(*
version 1.0	6 oct 2006
programmer 	hugo
tested by		tobias

findB_noNum searches str backwards and returns the last position which is not a number.
a number is characterized by a letter "0..9" or "."

*)
pt := ADR(str) + LEN(str) - 1;
findB_nonum := 0;
FOR pos := LEN(str) TO 1 BY -1 DO;
	IF NOT((PT^ > 47 AND PT^ < 58) OR PT^ = 46) THEN
		findB_nonum := pos;
		RETURN;
	END_IF;
	PT := PT - 1;
END_FOR;
END_FUNCTION

(* POU findB_Num, ST *)
FUNCTION findB_Num : INT
VAR_INPUT
	str : STRING;
END_VAR
VAR
	pos: INT;
	pt : POINTER TO BYTE;
END_VAR

(*
version 1.0	6 oct 2006
programmer 	hugo
tested by		tobias

findB_Num searches str backward and returns the last position of a number
a number is characterized by a letter "0..9" or "."

*)
pt := ADR(str) + LEN(str) - 1;
findB_Num := 0;
FOR pos := LEN(str) TO 1 BY -1 DO;
	IF (PT^ > 47 AND PT^ < 58) OR PT^ = 46 THEN
		findB_Num := pos;
		RETURN;
	END_IF;
	PT := PT - 1;
END_FOR;
END_FUNCTION

(* POU F_Lamp, ST *)
FUNCTION_BLOCK F_Lamp
VAR_INPUT
	SWITCH : BOOL;
	DIMM : BYTE := 255;
	Rst : BOOL;
END_VAR
VAR_OUTPUT
	Lamp : BYTE;
	ontime : REAL;
	cycles : REAL;
	Status : BYTE;
END_VAR
VAR_INPUT CONSTANT
	T_no_Dimm : REAL := 100;
	T_Maintenance : REAL := 15000;
END_VAR
VAR
	runtime : ontime;
	maintenance: BOOL;
END_VAR

(*
version 1.1	8 Feb 2007
programmer 	hugo
tested by		tobias

F_Lamp is an interface to flourescent lamps. its main purpose is to protect flourescent lamps from dimming within the first T_NO_DIMM Time.
If Flourescent Lamps are dimmed during the first 100 hours the lifetime of the lamp is reduced dramatically.
The interface also counts ontime and cycles of the lamp for maintanance purposes.

*)
IF rst THEN
	runtime.rst := TRUE;
	runtime();
	runtime.rst := FALSE;
	ontime := runtime.ontime;
	cycles := runtime.cycles;
	maintenance := FALSE;
ELSE
	runtime(in := Switch);
	ontime := runtime.ontime;
	cycles := runtime.cycles;
END_IF;

IF NOT maintenance AND runtime.ontime >= T_maintenance AND T_Maintenance > 0 THEN
	status := 120;
	maintenance := TRUE;
ELSIF Switch THEN
	IF runtime.ontime < T_no_Dimm THEN
		Lamp := 255;
		STATUS := 111;
	ELSE
		Lamp := DIMM;
		status := 112;
	END_IF;
ELSE
	lamp := 0;
	status := 110;
END_IF;
END_FUNCTION_BLOCK

(* POU F_lin, ST *)
FUNCTION F_lin : REAL
VAR_INPUT
	X : REAL;
	A : REAL;
	B : REAL;
END_VAR
VAR
END_VAR

(*
version 1.0	1 sep 2006
programmer 	hugo
tested by		tobias

this function calculates the linear equation f_lin = a*x + b

*)
F_lin := A * X + B;
END_FUNCTION

(* POU F_Lin2, ST *)
FUNCTION F_Lin2 : REAL
VAR_INPUT
	X : REAL;
	X1: REAL;
	Y1 : REAL;
	X2 : REAL;
	Y2 : REAL;
END_VAR
VAR

END_VAR

(*
version 1.0	1 jan 2007
programmer 	hugo
tested by		tobias

this function calculates the linear equation f_lin = a*x + b given by two points x1/y1 and x2/y2.

*)
F_Lin2 := (Y2 - Y1) / (X2 - X1) * X + (Y1 * X1 - Y2 * X1) / (X2 - X1) + Y1;
END_FUNCTION

(* POU F_power, ST *)
FUNCTION F_power : REAL
VAR_INPUT
	a : REAL;
	x : REAL;
	n : REAL;
END_VAR
VAR
END_VAR

(*
version 1.0	1 sep 2006
programmer 	hugo
tested by		tobias

this function calculates the power equation f_power = a*x^n

*)
f_power := a * EXPT(X,N);
END_FUNCTION

(* POU F_quad, ST *)
FUNCTION F_quad : REAL
VAR_INPUT
	X : REAL;
	A : REAL;
	B : REAL;
	C : REAL;
END_VAR
VAR
END_VAR

(*
version 1.0	1 sep 2006
programmer 	hugo
tested by		tobias

this function calculates the quadratic equation f_lin = a*x + b

*)
F_quad := a * X * X + B * X + C;
END_FUNCTION

(* POU F_to_C, ST *)
FUNCTION F_to_C : REAL
VAR_INPUT
	fahrenheit : REAL;
END_VAR
VAR
END_VAR

(*
version 1.0	4 aug 2006
programmer 	hugo
tested BY		tobias

this FUNCTION converts fahrenheit TO celsius

executioin TIME on wago 750-841 = 15us
*)
F_to_C := (fahrenheit -32) / 1.8;
END_FUNCTION

(* POU F_to_OM, ST *)
FUNCTION F_to_OM : REAL
VAR_INPUT
	F : REAL;
END_VAR
VAR
END_VAR

(*
version 1.0	22 jan 2007
programmer 	hugo
tested by		tobias

this function converts frequency to Omega F
Omega = 2*PI*F
*)
F_to_OM := PI2 * F;
END_FUNCTION

(* POU F_to_PT, ST *)
FUNCTION F_to_PT : TIME
VAR_INPUT
	F : REAL;
END_VAR
VAR
END_VAR

(*
version 1.0	4 aug 2006
programmer 	hugo
tested by		tobias

this function converts frequency to periode time  
*)
F_to_PT := DWORD_TO_TIME(REAL_TO_DWORD(1/F*1000));
END_FUNCTION

(* POU fact, ST *)
FUNCTION fact : INT
VAR_INPUT
	X : INT;
END_VAR
VAR
	i: INT;
END_VAR

(*
version 1.1	4 mar 2007
programmer 	hugo
tested by		tobias

this function calculates the factorial of x
this simple factorial only calculates factorials for inputs up to 7
if the input is negative or higher then 7 the output will be -1.

*)
IF x >= 0 AND x < 8 THEN
	fact := 1;
	i := 1;
	WHILE i <= x DO
		fact := fact * i;
		i := i + 1;
	END_WHILE;
ELSE
	fact := -1;
END_IF;

(* revision history
hm 4.3.2007	rev 1.1
	changed a critical error where while loop was indefinite.

*)
END_FUNCTION

(* POU FF_D2E, ST *)
FUNCTION_BLOCK FF_D2E
VAR_INPUT
	D0 : BOOL := 0;
	D1 : BOOL := 0;
	CLK : BOOL;
	RST : BOOL := 0;
END_VAR
VAR_OUTPUT
	Q0 : BOOL := 0;
	Q1 : BOOL := 0;
END_VAR
VAR
	edge : BOOL;
END_VAR

(*
version 1.0	4 aug 2006
programmer 	hugo
tested by		tobias

dual D-type flip flop with reset and rising clock trigger

executioin TIME on wago 750-841 = 6us
*)
IF rst THEN
	Q0 := FALSE;
	Q1 := FALSE;
ELSE
	IF clk AND NOT edge THEN
		Q0 := D0;
		Q1 := D1;
	END_IF;
END_IF;
edge := CLK;
END_FUNCTION_BLOCK

(* POU FF_D4E, ST *)
FUNCTION_BLOCK FF_D4E
VAR_INPUT
	D0 : BOOL := 0;
	D1 : BOOL := 0;
	D2 : BOOL := 0;
	D3 : BOOL := 0;
	CLK : BOOL;
	RST : BOOL := 0;
END_VAR
VAR_OUTPUT
	Q0 : BOOL := 0;
	Q1 : BOOL := 0;
	Q2 : BOOL := 0;
	Q3 : BOOL := 0;
END_VAR
VAR
	edge : BOOL;
END_VAR


(*
version 1.0	4 aug 2006
programmer 	hugo
tested by		tobias

quad D-type flip flop with reset and rising clock trigger

executioin TIME on wago 750-841 = 6us
*)
IF rst THEN
	Q0 := FALSE;
	Q1 := FALSE;
	Q2 := FALSE;
	Q3 := FALSE;
ELSE
	IF clk AND NOT edge THEN
		Q0 := D0;
		Q1 := D1;
		Q2 := D2;
		Q3 := D3;
	END_IF;
END_IF;
edge := CLK;
END_FUNCTION_BLOCK

(* POU FF_DRE, ST *)
FUNCTION_BLOCK FF_DRE
VAR_INPUT
	SET : BOOL;
	D : BOOL;
	CLK : BOOL;
	RST : BOOL;
END_VAR
VAR_OUTPUT
	Q : BOOL := 0;
END_VAR
VAR
	edge : BOOL;
END_VAR


(*
version 1.0	4 aug 2006
programmer 	hugo
tested by		tobias

D-type flip flop with set, reset and rising clock trigger
executioin TIME on wago 750-841 = 8us
*)
IF rst THEN
	Q := FALSE;
ELSIF set AND NOT rst THEN
	Q := TRUE;
ELSE
	IF clk AND NOT edge THEN Q := D; END_IF;
END_IF;
edge := CLK;
END_FUNCTION_BLOCK

(* POU FF_JKE, ST *)
FUNCTION_BLOCK FF_JKE
VAR_INPUT
	SET : BOOL;
	J : BOOL;
	CLK : BOOL;
	K : BOOL;
	RST : BOOL;
END_VAR
VAR_OUTPUT
	Q : BOOL := 0;
END_VAR
VAR
	edge : BOOL;
END_VAR


(*
version 1.0	4 aug 2006
programmer 	hugo
tested by		tobias

JK-type flip flop with set, reset and rising clock trigger
set and reset are asynchron while the FF is rising edge triggered
J=0 and K=0 and CLK >>> no action
J=1 and K=0 and CLK >>> output = 1
J=0 and K=1 and CLK >>> output = 0
J=1 and K=1 and CLK >>> toggle output

executioin TIME on wago 750-841 = 8us
*)
IF rst THEN
	Q := FALSE;
ELSIF set AND NOT rst THEN
	Q := TRUE;
ELSE
	IF clk AND NOT edge THEN
		IF J AND NOT K THEN Q := TRUE;
		ELSIF K AND NOT J THEN Q := FALSE;
		ELSIF K AND J THEN Q:= NOT Q;
		END_IF;
	END_IF;
END_IF;
edge := CLK;
END_FUNCTION_BLOCK

(* POU FIFO_16, ST *)
FUNCTION_BLOCK FIFO_16
VAR_INPUT
	Din : DWORD;
	WR : BOOL;
	E : BOOL;
	RST : BOOL;
END_VAR
VAR_OUTPUT
	Dout : DWORD := 0;
	empty : BOOL := TRUE;
	full : BOOL := FALSE;
END_VAR
VAR
	fifo : ARRAY[0..15] OF DWORD;
	NW : INT := 0;
	NR : INT := 0;
	top : INT := 15;
END_VAR

(*
	version 1.0	4 aug 2006
	programmer 	hugo
	tested by		tobias

16 Dword FIFO memory
*)
IF rst THEN
	(* asynchronous reset for the fifo *)
	NW := 0;
	NR := 0;
	Dout := 0;
	empty := TRUE;
	full := FALSE;
ELSIF WR AND E AND NOT full THEN
	(* write action *)
	fifo[NW] := Din;
	IF NW = top THEN NW := 0; ELSE NW := NW + 1; END_IF
	IF NW = NR THEN full := TRUE; END_IF
	empty := FALSE;
ELSIF NOT WR AND E AND NOT empty THEN
	(* read from stack *)
	Dout := fifo[NR];
	IF NR = top THEN NR := 0; ELSE NR := NR + 1; END_IF;
	IF NR = NW THEN empty := TRUE; END_IF;
	full := FALSE;
END_IF;
END_FUNCTION_BLOCK

(* POU FIFO_32, ST *)
FUNCTION_BLOCK FIFO_32
VAR_INPUT
	Din : DWORD;
	WR : BOOL;
	E : BOOL;
	RST : BOOL;
END_VAR
VAR_OUTPUT
	Dout : DWORD := 0;
	empty : BOOL := TRUE;
	full : BOOL := FALSE;
END_VAR
VAR
	fifo : ARRAY[0..31] OF DWORD;
	NW : INT := 0;
	NR : INT := 0;
	top : INT := 31;
END_VAR

(*
	version 1.0	4 aug 2006
	programmer 	hugo
	tested by		tobias

32 Dword FIFO memory
*)
IF rst THEN
	(* asynchronous reset for the fifo *)
	NW := 0;
	NR := 0;
	Dout := 0;
	empty := TRUE;
	full := FALSE;
ELSIF WR AND E AND NOT full THEN
	(* write action *)
	fifo[NW] := Din;
	IF NW = top THEN NW := 0; ELSE NW := NW + 1; END_IF
	IF NW = NR THEN full := TRUE; END_IF
	empty := FALSE;
ELSIF NOT WR AND E AND NOT empty THEN
	(* read from stack *)
	Dout := fifo[NR];
	IF NR = top THEN NR := 0; ELSE NR := NR + 1; END_IF;
	IF NR = NW THEN empty := TRUE; END_IF;
	full := FALSE;
END_IF;
END_FUNCTION_BLOCK

(* POU find_nonum, ST *)
FUNCTION find_nonum : INT
VAR_INPUT
	str : STRING;
END_VAR
VAR
	pos: INT;
	pt : POINTER TO BYTE;
END_VAR

(*
version 1.0	6 oct 2006
programmer 	hugo
tested by		tobias

find_noNum searches str and returns the first position which is not a number.
a number is characterized by a letter "0..9" or "."

*)
pt := ADR(str);
find_nonum := 0;
FOR pos := 1 TO LEN(str) DO;
	IF NOT((PT^ > 47 AND PT^ < 58) OR PT^ = 46) THEN
		find_nonum := pos;
		RETURN;
	END_IF;
	PT := PT + 1;
END_FOR;
END_FUNCTION

(* POU find_Num, ST *)
FUNCTION find_Num : INT
VAR_INPUT
	str : STRING;
END_VAR
VAR
	pos: INT;
	pt : POINTER TO BYTE;
END_VAR

(*
version 1.0	6 oct 2006
programmer 	hugo
tested by		tobias

find_Num searches str and returns the starting position of a number
a number is characterized by a letter "0..9" or "."

*)
pt := ADR(str);
find_Num := 0;
FOR pos := 1 TO LEN(str) DO;
	IF (PT^ > 47 AND PT^ < 58) OR PT^ = 46 THEN
		find_Num := pos;
		RETURN;
	END_IF;
	PT := PT + 1;
END_FOR;
END_FUNCTION

(* POU FindB, ST *)
FUNCTION FindB : INT
VAR_INPUT
	str1 : STRING;
	str2 : STRING;
END_VAR
VAR
	pos: INT;
	size: INT;
	length: INT;
END_VAR

(*
version 1.0	6 oct 2006
programmer 	hugo
tested by		tobias

the function find searches an str1 for the presence of str2 and returns the first position of str1 of the last presence in instring.
the function is similar to find except it searches from the right to left.
 a 0 is returned if the string is not found.

*)
size := LEN(str1);
length := LEN(str2);
FOR pos := size TO 1 BY -1 DO
	IF MID(str1,length,pos) = str2 THEN
		FindB := pos;
		RETURN;
	END_IF;
END_FOR;
END_FUNCTION

(* POU floor, ST *)
FUNCTION floor : INT
VAR_INPUT
	X : REAL;
END_VAR
VAR
END_VAR


(*
version 1.0	7 feb 2007
programmer 	hugo
tested by		tobias

This is a rounding function which returns the biggest possible integer which is less or equal to X.
floor(3.14) = 3
floor(-3.14) = 4

*)
floor := TRUNC(X);
IF floor > X THEN
	floor := floor - 1;
END_IF;
END_FUNCTION

(* POU fract, ST *)
FUNCTION fract : REAL
VAR_INPUT
	input : REAL;
END_VAR
VAR
END_VAR
VAR
END_VAR

(*
version 1.0	4 aug 2006
programmer 	hugo
tested by		tobias

this function returns the fraction of a real number
fract(3.14) = 0.14

execution time on wago 750 - 841 =  17  us
*)
fract := input - TRUNC(input);
END_FUNCTION

(* POU FT_avg, ST *)
FUNCTION_BLOCK FT_avg
VAR_INPUT
	in : REAL;
	en : BOOL;
	N : INT;
	rst : BOOL;
END_VAR
VAR_OUTPUT
	avg : REAL;
END_VAR
VAR
	buff : delay;
	i: INT;
	init : BOOL;
END_VAR

(*
version 1.1	7 jan 2007
programmer 	hugo
tested by		tobias

this function calculates the average over n samples from a sequential input
the input values are shifted into an N deep buffer and the avg of this buffer is diplayed at anytime on the output.
a rst will load the buffer with the current in value..

*)
(* limit n to a max of 32 because delay can do max 32 cycles *)
IF N > 32 THEN
	buff.n := 32;
ELSIF N < 0 THEN
	Buff.n := 0;
ELSE
	buff.n := N;
END_IF;

IF NOT init THEN
	FOR i := 1 TO N DO
		buff(in := in);
	END_FOR;
	avg := in;
	init := TRUE;
ELSIF rst THEN
	FOR i := 1 TO N DO
		buff(in := in);
	END_FOR;
	avg := in;
ELSIF en THEN
	buff(in := in);
	avg := avg + (in - buff.out)/N;
END_IF;

(* revision history

hm	7.1.2007	rev 1.1
	chaged rst logic to load the buffer with the actual input value instead of 0.
	added en input to allow better control of signal flow
	added init to load the buffer with inat startup to avoid rampup at beginning.
	deleted unused variable cnt.
*)
END_FUNCTION_BLOCK

(* POU FT_deriv, ST *)
FUNCTION_BLOCK FT_deriv
VAR_INPUT
	in : REAL;
	K : REAL := 1;
	run : BOOL := 1;
END_VAR
VAR_OUTPUT
	out : REAL;
END_VAR
VAR
	old: REAL;
	tx: TIME;
	last: TIME;
	init: BOOL;
END_VAR


(*
version 1.1	3 jan 2007
programmer 	hugo
tested by		tobias

FT_deriv calculates the derivate over the signal "in" with Faktor "K".
a run input enables or stops the calculation, if left unconnected its true and therfore the calculation is executed.
if K is not specified the default is 1.

*)
tx := TIME();
IF NOT init THEN
	init := TRUE;
	old := in;
	last := tx;
END_IF;
IF run THEN
	out := (in - old) / TIME_TO_REAL(tx - last) * 1000 * K;
ELSE
	out := 0;
END_IF;
old := in;
last := tx;

(*
hm 3.1.2007	rev 1.1
	added init code for startup
	set the default for K to 1

*)
END_FUNCTION_BLOCK

(* POU FT_IMP, ST *)
FUNCTION_BLOCK FT_IMP
VAR_INPUT
	in : REAL;
	T : TIME;
	K : REAL := 1;
END_VAR
VAR_OUTPUT
	out : REAL;
END_VAR
VAR
	t1 : FT_PT1;
END_VAR

(*
version 1.1	3 Jan 2007
programmer 	hugo
tested by		tobias

FT_IMP is 	an impulse filter (high pass filter) with the time T and factor K.
 
*)
T1(in:= in, T:=T);
out := (in - t1.out) * K;

(*
hm 3.1.2007	rev 1.1
	added factor K

*)
END_FUNCTION_BLOCK

(* POU FT_PT1, ST *)
FUNCTION_BLOCK FT_PT1
VAR_INPUT
	in : REAL;
	T : TIME;
	K : REAL := 1;
END_VAR
VAR_OUTPUT
	out : REAL;
END_VAR
VAR
	last : TIME;
	tx: TIME;
	init: BOOL;
END_VAR

(*
version 1.3	27 feb 2007
programmer 	hugo
tested by		tobias

FT_PT1 is an low pass filter with a programmable time T and faktor K.
 
*)
tx := TIME();
IF NOT init THEN
	last := tx;
	init := TRUE;
ELSIF T = t#0s THEN
	out := in;
ELSE
	out := out + (in * K - out) * TIME_TO_REAL(Tx - last) / TIME_TO_REAL(T);
END_IF;
last := tx;

(*
hm 1.1.2007	rev 1.1
	corrected error while startup value was not correct
	for very small time values real output would run out of range.

hm 3.1.2007	rev 1.2
	corrected an error for falling edge failures.
	added output faktor K.

hm 27. 2. 2007	rev 1.3
	output will be input during init for definitive startup condition.
*)
END_FUNCTION_BLOCK

(* POU FT_INT, ST *)
FUNCTION_BLOCK FT_INT
VAR_INPUT
	in : REAL;
	K : REAL := 1;
	run : BOOL := 1;
	rst: BOOL := 0;
	out_min : REAL := -1000;
	out_max : REAL := 1000;
END_VAR
VAR_OUTPUT
	Out : REAL;
	ET: TIME;
END_VAR
VAR
	last: TIME;
	in_last : REAL;
	tx: TIME;
	init: BOOL;
END_VAR


(*
version 1.2	15 jan 2007
programmer 	hugo
tested by		tobias

FT_int is an integrator with input IN and factor K.
integration is only done while run = true, if run is false integration is stopped and the out remains at the last value.
if run is left unconnected, run is considered true by the function block.
the output ET will display the total integration time from last reset.
a rst input will reset output and the timer ET to 0.
the out_min and out_max values can be set to ,imit the output value range. 
out _min is preset to -1000 and out_max is preset to 1000.
the default for K is 1.

 
*)
last := tx;
tx := TIME();
IF rst OR NOT init THEN
	out := 0;
	ET := t#0s;
	init := TRUE;
	last := tx;
ELSIF run THEN
	out := out + (in + in_last)/2 * TIME_TO_DINT(Tx-last) * K / 1000;
	IF out < out_min THEN out := out_min; ELSIF out > out_max THEN out := out_max; END_IF;
	et := et + Tx - last;
END_IF;
in_last := in;

(*
hm 13.12.2006	rev 1.1
changed to "trapezregel" which increases accuracy
before out := out + in * time new: out := out + (in + in_last) / 2 * time

hm 15.1.2007		rev 1.2
added default for k to be 1.
*)
END_FUNCTION_BLOCK

(* POU FT_min_max, ST *)
FUNCTION_BLOCK FT_min_max
VAR_INPUT
	in : REAL;
	rst : BOOL;
END_VAR
VAR_OUTPUT
	mx : REAL;
	mn : REAL;
END_VAR
VAR
	init: BOOL;
END_VAR

(*
version 1.0	1 sep 2006
programmer 	hugo
tested by		tobias

this function block stores the min and max value of an input signal.
when rst is true the mn and mx outputs are set to the in value.
when a rst is never active the function autoresets to the in value at startup.
since the input might not be present at first cycle the mn and mx are set during second cycle.

*)
IF rst OR NOT init THEN
	mn := in;
	mx := in;
	init := 1;
ELSIF in < mn THEN mn := in;
ELSIF in > mx THEN mx := in;
END_IF;
END_FUNCTION_BLOCK

(* POU FT_PID, ST *)
FUNCTION_BLOCK FT_PID
VAR_INPUT
	actual, set_point, offset, manual_in : REAL;
	Manual : BOOL;
	rst : BOOL := FALSE;
	int_band : REAL := 100;
END_VAR
VAR_INPUT
	KP : REAL := 1.0;
	TN : REAL := 1.0;
	TV : REAL := 1.0;
	limit_L : REAL := -1000;
	limit_H : REAL := 1000;
END_VAR
VAR_OUTPUT
	Y : REAL;
	LIM, overflow : BOOL;
END_VAR
VAR
	integ : FT_INT;
	deriv : FT_deriv;
	diff: REAL;
END_VAR

(*
version 1.3	3 mar 2007
programmer 	hugo
tested by		tobias

FT_PID is a pid controller with manual functionality.
The PID controller works according to the fomula Y = KP * ( e + 1/TN * INTEG(e) + TV *DERIV(e)) + offset, while e = set_point - actual.
a rst will reset all internal data, while a switch to manual will cause the controller to follow the function Y = manual_in + offset.
limit_h and Limit_l set the possible output range of Y.
the output flags lim will signal that the output limits are active and overflow will signal that the integrator has reached the max or min limit.  

since rev 1.1 the "trapezregel is used for more accuracy.
rev 1.2 added selective integratin which means the integrative component is only active within a small range of the target value 
this avoids the integrator to go to limits while an input setpoint change happened and is only causing overshoots.
the int_band is by default 100 which means the int is active all the time and if set to for example to 0.1 the integrator is only active
while the input is between 0.9 and 1.1 of the set_point value.

default values for KP = 1, TN = 1, TV = 1, LIMIT_L = -1000, LIMIT_H = +1000.
*)
IF rst OR KP = 0 THEN
	y := offset;
	integ(rst := 1);
	integ.rst := 0;
ELSIF manual THEN
	Y := manual_in + offset;
	integ(rst := 1);
	integ.rst := 0;
ELSE
	(* calcualtion of the actual PID values *)
	diff := set_point - actual;

	(* integrator is only called if TN > 0 and input is within int_band othewrwise it is disabled *)
	IF TN > 0 AND actual > set_point - int_band AND actual < set_point + int_band THEN
		integ(in := diff, K := 1/TN, out_min := (limit_L - offset) / KP, out_max := (limit_H - offset) / KP);
	ELSE
		integ(rst := 1);
		integ.rst := 0;
	END_IF;
	deriv(in := diff, K := TV);

	(* check if integrator has reached the allowed limits and set overflow if necessary *)
	IF integ.Out >= (limit_H - offset) / KP THEN
		Y := limit_H;
		overflow := TRUE;
	ELSIF integ.Out <= (limit_L - offset) / KP THEN
		Y := limit_L;
		overflow := TRUE;
	ELSE
		Y := KP * (integ.Out + deriv.out + diff) + offset;
		overflow := FALSE;
	END_IF;

	(* this portion limits the output to limit_H and limit_L and set the lim flag if limits are exceeded *)
	IF Y > limit_H THEN
		Y := limit_H;
		Lim := TRUE;
	ELSIF Y < limit_L THEN
		Y := limit_L;
		lim := TRUE;
	ELSE
		lim := FALSE;
	END_IF;
END_IF;

(* revision history

hm 1.12.2006 rev 1.1
	changed algorithm to trapezregel for higher accuracy.

hm 3.1.2007	rev 1.2
	added integ_band to select when the integrator is active.

hm	3.3.2007	rev 1.3
	added default values to inputs KP, TN, TV, LIMIT_L und LIMIT_H.

*)
END_FUNCTION_BLOCK

(* POU FT_Profile, ST *)
FUNCTION_BLOCK FT_Profile
VAR_INPUT
	K : REAL := 1;
	O : REAL := 0;
	M : REAL := 1;
	E : BOOL;
END_VAR
VAR_INPUT CONSTANT
	value_0 : REAL;
	time_1 : TIME;
	value_1 : REAL;
	time_2 : TIME;
	value_2 : REAL;
	time_3 : TIME;
	value_3 : REAL;
	time_10 : TIME;
	value_10 : REAL;
	time_11 : TIME;
	value_11 : REAL;
	time_12 : TIME;
	value_12 : REAL;
	time_13 : TIME;
	value_13 : REAL;
END_VAR
VAR_OUTPUT
	Y : REAL;
	RUN : BOOL;
	ET : TIME;
END_VAR
VAR
	tx : TIME;
	edge : BOOL;
	state: BYTE;
	ta: TIME;
	tb: TIME;
	t0 : TIME;
	temp: REAL;
	va: REAL;
	vb: REAL;
END_VAR

(*
version 1.0	27 feb 2007
programmer 	tobias
tested by		hugo

FT_Profile generates an output signal which is defined by values over a time scale.
the different values are connected by ramps between the individual values.
a rising edge on E starts the output signal generation and E = True can delay time_3 / value_3 as long as it stays true.
an additional multiplier K can be used to multiply the output and an offset O can be added to the output dynamically.
*)
(* read system time *)
tx := TIME();

(* determine start condition *)
IF E AND NOT edge THEN
	RUN := TRUE;
	ET := t#0s;
	t0 := tx;
	ta := tx;
	tb := multime(time_1, M);
	va := value_0;
	vb := value_1;
	temp := value_0;
	state := 1;
END_IF;
edge := E;

(* generate startup profile *)
IF run THEN
	CASE state OF
		1:	IF tx - ta >= tb THEN
				ta := ta + tb;
				tb := multime(time_2 - time_1, M);
				va := value_1;
				vb := value_2;
				temp := value_1;
				state := 2;
			ELSE
				temp := ((vb - va) * TIME_TO_REAL(tx - ta) / TIME_TO_REAL(tb) + va);
			END_IF;
		2:	IF tx - ta >= tb THEN
				ta := ta + tb;
				tb := multime(time_3 - time_2, M);
				va := value_2;
				vb := value_3;
				temp := value_2;
				state := 3;
			ELSE
				temp := ((vb - va) * TIME_TO_REAL(tx - ta) / TIME_TO_REAL(tb) + va);
			END_IF;
		3:	IF tx - ta >= tb THEN
				ta := ta + tb;
				tb := multime(time_10 - time_3, M);
				va := value_3;
				vb := value_10;
				temp := value_3;
				state := 4;
			ELSE
				temp := ((vb - va) * TIME_TO_REAL(tx - ta) / TIME_TO_REAL(tb) + va);
			END_IF;
		4 :	IF tx - ta >= tb THEN
				ta := ta + tb;
				tb := multime(time_11 - time_10, M);
				va := value_10;
				vb := value_11;
				temp := value_10;
				IF E THEN state := 5; ELSE state := 6; END_IF;
			ELSE
				temp := ((vb - va) * TIME_TO_REAL(tx - ta) / TIME_TO_REAL(tb) + va);
			END_IF;
		5:	(* extend the signal while E is true *)
			IF E THEN
				ta := tx;
			ELSE
				state := 6;
			END_IF;
		6:	IF tx - ta >= tb THEN
				ta := ta + tb;
				tb := multime(time_12 - time_11, M);
				va := value_11;
				vb := value_12;
				temp := value_11;
				state := 7;
			ELSE
				temp := ((vb - va) * TIME_TO_REAL(tx - ta) / TIME_TO_REAL(tb) + va);
			END_IF;
		7:	IF tx - ta >= tb THEN
				ta := ta + tb;
				tb := multime(time_13 - time_12, M);
				va := value_12;
				vb := value_13;
				temp := value_12;
				state := 8;
			ELSE
				temp := ((vb - va) * TIME_TO_REAL(tx - ta) / TIME_TO_REAL(tb) + va);
			END_IF;
		8:	IF tx - ta >= tb THEN
				temp := value_13;
				run := FALSE;
			ELSE
				temp := ((vb - va) * TIME_TO_REAL(tx - ta) / TIME_TO_REAL(tb) + va);
			END_IF;
	END_CASE;
	Y := temp * K + O;
	ET := tx - t0;
END_IF;
END_FUNCTION_BLOCK

(* POU FT_PT2, ST *)
FUNCTION_BLOCK FT_PT2
VAR_INPUT
	in : REAL;
	T : TIME;
	D : REAL;
	K : REAL := 1;
END_VAR
VAR_OUTPUT
	out : REAL;
END_VAR
VAR
	last : TIME;
	tx: TIME;
	init: BOOL;
	int1 : FT_INT;
	int2 : FT_INT;
	tn: REAL;
END_VAR

(*
version 1.1	15 jan 2007
programmer 	hugo
tested by		tobias

FT_PT2 is a 2nd grade filter with programmable times T, D and faktor K.
 
*)
last := tx;
tx := TIME();
IF NOT init THEN
	last := tx;
	out :=in;
	init := TRUE;
ELSE
	TN := TIME_TO_REAL(T)/1000;
	int1(in := in * K / (TN * TN) - int1.Out * 2 *D / TN - int2.Out / (TN * TN));
	int2(in := int1.Out);
	out := int2.out;
END_IF;

(* revision history

15.1.2007 hm		rev 1.1
	changed formula to new more acurate formula
	old code:
	tx := TIME();
	IF NOT init THEN
		last := tx;
		init := TRUE;
	ELSE
		IF T> t#0s THEN
			out1 := out1 + (in - out1) * TIME_TO_REAL(Tx - last) / TIME_TO_REAL(T);
		ELSE
			out1 := in;
		END_IF;
		IF T > t#0s THEN
			out2 := out2 + (out1 - out2) * TIME_TO_REAL(Tx - last) / TIME_TO_REAL(T);
		ELSE
			out2 := out1;
		END_IF;
		out := out2 * K;
	END_IF;
	last := tx;

*)
END_FUNCTION_BLOCK

(* POU FT_TN16, ST *)
FUNCTION_BLOCK FT_TN16
VAR_INPUT
	in : REAL;
	T : TIME;
END_VAR
VAR_OUTPUT
	out : REAL;
	trig : BOOL;
END_VAR
VAR
	length : INT := 16;
	X : ARRAY[0..15] OF REAL;
	cnt : INT;
	last : TIME;
	tx: TIME;
	init: BOOL;
END_VAR

(*
version 1.0	1 Jan 2007
programmer 	hugo
tested by		tobias

FT_TN16 is delay function, it will delay a signal by a specified time : T and will store 16 values of in before they are put thru to out.
for higher or lower resolution please use FT_TN8 or FT_TN64 instead.
 
*)
tx := TIME();
trig := FALSE;
IF NOT init THEN
	x[cnt] := in;
	init := TRUE;
	last := tx;
ELSIF tx - last >= T / length THEN
	IF cnt = length - 1 THEN cnt := 0; ELSE cnt := cnt + 1; END_IF;
	Out := X[cnt];
	x[cnt] := in;
	last := tx;
	Trig := TRUE;
END_IF;
END_FUNCTION_BLOCK

(* POU FT_TN64, ST *)
FUNCTION_BLOCK FT_TN64
VAR_INPUT
	in : REAL;
	T : TIME;
END_VAR
VAR_OUTPUT
	out : REAL;
	trig: BOOL;
END_VAR
VAR
	length : INT := 64;
	X : ARRAY[0..63] OF REAL;
	cnt : INT;
	last : TIME;
	tx: TIME;
	init: BOOL;
END_VAR

(*
version 1.0	1 Jan 2007
programmer 	hugo
tested by		tobias

FT_TN7 is delay function, it will delay a signal by a specified time : T and will store 64 values of in before they are put thru to out.
if lower resolution is needed, pls use FT_TN8 or FT_TN16 instead.
 
*)
tx := TIME();
trig := FALSE;
IF NOT init THEN
	x[cnt] := in;
	init := TRUE;
	last := tx;
ELSIF tx - last >= T / length THEN
	IF cnt = length - 1 THEN cnt := 0; ELSE cnt := cnt + 1; END_IF;
	Out := X[cnt];
	x[cnt] := in;
	last := tx;
	trig := TRUE;
END_IF;
END_FUNCTION_BLOCK

(* POU FT_TN8, ST *)
FUNCTION_BLOCK FT_TN8
VAR_INPUT
	in : REAL;
	T : TIME;
END_VAR
VAR_OUTPUT
	out : REAL;
	trig: BOOL;
END_VAR
VAR
	length : INT := 8;
	X : ARRAY[0..7] OF REAL;
	cnt : INT;
	last : TIME;
	tx: TIME;
	init: BOOL;
END_VAR

(*
version 1.0	1 Jan 2007
programmer 	hugo
tested by		tobias

FT_TN8 is delay function, it will delay a signal by a specified time : T and will store 8 values of in before they are put thru to out.
if higher resolution is needed, pls use FT_TN16 or FT_TN64 instead.
 
*)
tx := TIME();
trig := FALSE;
IF NOT init THEN
	x[cnt] := in;
	init := TRUE;
	last := tx;
ELSIF tx - last >= T / length THEN
	IF cnt = length - 1 THEN cnt := 0; ELSE cnt := cnt + 1; END_IF;
	Out := X[cnt];
	x[cnt] := in;
	last := tx;
	trig := TRUE;
END_IF;
END_FUNCTION_BLOCK

(* POU gen_bit, ST *)
FUNCTION_BLOCK gen_bit
VAR_INPUT
	in0 : DWORD;
	in1 : DWORD;
	in2 : DWORD;
	in3 : DWORD;
	clk : BOOL := 0;
	steps : INT;
	rep : INT := 0;
	rst : BOOL := 0;
END_VAR
VAR_OUTPUT
	Q0 :BOOL := 0;
	Q1 :BOOL := 0;
	Q2 :BOOL := 0;
	Q3 :BOOL := 0;
	cnt : INT := 0;
	run : BOOL := 0;
END_VAR
VAR
	r0: DWORD;
	r1: DWORD;
	r2: DWORD;
	r3: DWORD;
	rx : INT := 1;
END_VAR

(*
version 1.0	4 aug 2006
programmer 	hugo
tested by		tobias

gen_bit is 4 bit sequencial pattern generator with 4 DWORD inputs and 4 serial outputs.
with the first clock pulse after a reset or after power on, bit 0 of the input DWORDS IN is present on the Outputs Q and the next clock cycle shifts to Bit 1 and so on.
the input steps defines how many bits of the input dwords will be shifted to the outputs. the sequence can be repetive when rep = 0 or any amount of repetitions can be defined with input rep.

*)
(* check if number of runs is finished or rep = 0 which means continuous *)

IF clk AND NOT rst THEN
	IF (rep = 0) OR (rx <= rep) THEN run := TRUE; ELSE run := FALSE; END_IF;
	IF run THEN
		(* check for step counter reached and reset to 0 if cnt = steps *)
		IF cnt = steps THEN
			cnt := 0;
		END_IF;

		(* when cnt = 0 then reload the inputs into the registers *)
		IF cnt = 0 THEN
			r0 := in0;
			r1 := in1;
			r2 := in2;
			r3 := in3;
		END_IF;

		(* when cnt < steps, shift the lowest bits to the outputs *)
		IF (cnt < steps) THEN
			Q0 := r0.0;
			Q1 := r1.0;
			Q2 := r2.0;
			Q3 := r3.0;
			r0 := SHR(r0,1);
			r1 := SHR(r1,1);
			r2 := SHR(r2,1);
			r3 := SHR(r3,1);
		END_IF;

		(* increment the step counter *)
		cnt := cnt +1;
		IF (cnt = steps) AND (rep <> 0) THEN rx := rx +1; END_IF;
		IF (rx > rep) AND (rep <> 0) THEN run := FALSE; END_IF;
	END_IF;
ELSE
	IF rst THEN
		Q0 := FALSE;
		Q1 := FALSE;
		Q2 := FALSE;
		Q3 := FALSE;
		r0 := 0;
		r1 := 0;
		r2 := 0;
		r3 := 0;
		cnt := 0;
		run := FALSE;
		rx := 1;
	END_IF;
END_IF;
END_FUNCTION_BLOCK

(* POU gen_rdm, ST *)
FUNCTION_BLOCK gen_rdm
VAR_INPUT
	PT : TIME;
	AM : REAL := 1;
	OS : REAL;
END_VAR
VAR_OUTPUT
	Q : BOOL;
	Out : REAL;
END_VAR
VAR
	tx : TIME;
	last : TIME;
	init : BOOL;
END_VAR

(*
	version 1.0	7 feb 2007
	programmer 	oscat
	tested BY		oscat

this signal generator generates a random output. The signal is defined by period time (PT), 
amplitude (AM), offset (OS).
The Output waveform will have its max peak at AM/2 + OS and its minimum peak at -AM/2 + OS. 
The period time PT defines how often the output signal will jump to a new randow value.
The Output Q will be true for one cycle anytime the output OUT has changed

*)
(* read system time and prepare input data *)
tx := TIME() - last;

(* init section *)
IF NOT init THEN
	init := TRUE;
	last := tx;
	tx := t#0s;
END_IF;

(* add last if one cycle is finished *)
IF tx >= pt THEN
	last := last + pt;
	tx := tx - pt;

	(* generate output signal *)
	out := am * (RDM(0) - 0.5) + os;
	q := TRUE;
ELSE
	q := FALSE;
END_IF;
END_FUNCTION_BLOCK

(* POU RDM, ST *)
FUNCTION RDM : REAL
VAR_INPUT
	last : REAL;
END_VAR
VAR
	temp: REAL;
END_VAR


(*
version 1.0	16 jan 2007
programmer 	hugo
tested by		tobias

this function calculates a pseudo random number
to generate the number it reads the sps timer and calculates a random number between 0 and 1:
in order to use rdm more then once within one sps cycle it need to be called with different seed numbers LAST.

*)
temp := TIME_TO_WORD(TIME());
RDM := fract(modR(temp*e, pi-last) + modR(temp*pi + last,e-last));
END_FUNCTION

(* POU modR, ST *)
FUNCTION modR : REAL
VAR_INPUT
	in : REAL;
	divi : REAL;
END_VAR
VAR
END_VAR
VAR
END_VAR

(*
version 1.1	4 aug 2006
programmer 	hugo
tested by		tobias

this is a modulo funtion for real numbers
modr(5.5,2.5) = 0.5


execution time on wago 750 - 841 =  29  us
*)
IF divi = 0 THEN
	modR := 0;
ELSE
	modR := in - TRUNC(in / divi)*divi;
END_IF;

(* revision history

hm 4.8.2006	rev 1.0

hm 28.1.2007	rev 1.1
	modr(x,0) will deliver the result 0

*)
END_FUNCTION

(* POU gen_rmp, ST *)
FUNCTION_BLOCK gen_rmp
VAR_INPUT
	PT : TIME := t#1s;
	AM : REAL := 1;
	OS : REAL := 0;
	DL : REAL := 0;
END_VAR
VAR_OUTPUT
	Q : BOOL;
	Out : REAL;
END_VAR
VAR
	tx : TIME;
	last : TIME;
	init : BOOL;
	temp : REAL;
	ltemp: REAL;
END_VAR

(*
	version 1.0	3 mar 2007
	programmer 	oscat
	tested BY		oscat

this signal generator generates a ramp wave output. The ramp wave signal is defined by period time (PT), 
amplitude (AM), offset (OS) and a specific delay for the output signal (DL).
The Output waveform will have its minimum peak at OS and its maximum peak at AM + OS. 
The delay input can delay a signal up to PT, this can be useful to synchronize different generators 
and generate interleaving signals.
in addition to the analog output Out there is a second boolean output Q with is true for one cycle when the ramp starts.
*)
(* read system time and prepare input data *)
tx := TIME() - last;
DL := modR(dl,1);
IF dl < 0 THEN dl := 1 - dl; END_IF;

(* init section *)
IF NOT init THEN
	init := TRUE;
	last := tx;
	tx := t#0s;
END_IF;

(* add last if one cycle is finished *)
IF tx >= pt THEN
	last := last + pt;
	tx := tx - pt;
END_IF;

(* generate sine wave *)
ltemp := temp;
temp := fract(TIME_TO_REAL(tx + multime(pt, dl)) / TIME_TO_REAL(pt));
out := am * temp + os;

(* boolean output Q *)
IF temp < ltemp THEN
	q := TRUE;
ELSE
	q := FALSE;
END_IF;
END_FUNCTION_BLOCK

(* POU gen_sin, ST *)
FUNCTION_BLOCK gen_sin
VAR_INPUT
	PT : TIME;
	AM : REAL := 1;
	OS : REAL;
	DL : REAL;
END_VAR
VAR_OUTPUT
	Q : BOOL;
	Out : REAL;
END_VAR
VAR
	tx : TIME;
	last : TIME;
	init : BOOL;
	temp : REAL;
END_VAR

(*
	version 1.0	22 jan 2007
	programmer 	oscat
	tested BY		oscat

this signal generator generates a sine wave output. The sine wave signal is defined by period time (PT), 
amplitude (AM), offset (OS) and a specific delay for the output signal (DL).
The Output waveform will have its max peak at AM/2 + OS and its minimum peak at -AM/2 + OS. 
The delay input can delay a signal up to PT, this can be useful to synchronize different generators 
and generate interleaving signals. A Cos wave can be generated accordingly.
in addition to a analog output Out there is a second boolean output Q with the corresponding binary signal.
*)
(* read system time and prepare input data *)
tx := TIME() - last;
DL := modR(dl,1);
IF dl < 0 THEN dl := 1 - dl; END_IF;

(* init section *)
IF NOT init THEN
	init := TRUE;
	last := tx;
	tx := t#0s;
END_IF;

(* add last if one cycle is finished *)
IF tx >= pt THEN
	last := last + pt;
	tx := tx - pt;
END_IF;

(* generate sine wave *)
temp := SIN(PI2 * TIME_TO_DWORD(tx + multime(pt, dl)) / TIME_TO_DWORD(pt));
out := am / 2 *  temp + os;

(* boolean output Q *)
q := NOT sign_R(temp);
END_FUNCTION_BLOCK

(* POU gen_SQ, ST *)
FUNCTION_BLOCK gen_SQ
VAR_INPUT
	PT : TIME := T#0ms;
END_VAR
VAR_OUTPUT
	Q : BOOL := 0;
END_VAR
VAR
	pti : TIME := t#0ms;
	run: BOOL := FALSE;
	next_edge: TIME := t#0ms;
	overflow: BOOL := 0;
END_VAR

(*
version 1.0	4 aug 2006
programmer 	hugo
tested by		tobias

gen_sq generates square wave signal with programmable period time.
the period time is defined for 10ms .. 65s
if the period time is set to less then 10ms the min perid is 10ms.

*)
IF NOT run THEN
	next_edge := TIME();
	run := TRUE;
	IF pt < T#10ms THEN PTI := T#5ms; ELSE pti := pt / 2; END_IF;
END_IF;
IF (TIME() >= next_edge) AND NOT overflow THEN
	Q := NOT Q;
	IF next_edge + pti < next_edge THEN
		(* time() will overflow every 50 days *)
		overflow := TRUE;
	END_IF;
	next_edge := next_edge + pti;
ELSE
	(* wait till time() has an overflow and reset overflow *)
	IF TIME() <= next_edge THEN overflow := FALSE; END_IF;
END_IF;
END_FUNCTION_BLOCK

(* POU gen_sqr, ST *)
FUNCTION_BLOCK gen_sqr
VAR_INPUT
	PT : TIME;
	AM : REAL;
	OS : REAL;
	DC : REAL := 0.5;
	DL : REAL;
END_VAR
VAR_OUTPUT
	Q : BOOL;
	Out : REAL;
END_VAR
VAR
	tx : TIME;
	last : TIME;
	init: BOOL;
END_VAR

(*
	version 1.1	12 feb 2007
	programmer 	oscat
	tested BY		oscat

this signal generator generates a square wave output. The square wave signal is defined by period time (PT), 
amplitude (AM), offset (OS), duty cycle (DC) and a specific delay for the output signal (DL).
The Output waveform will switch between AM/2 + OS and -AM/2 + OS. The DC input specifies ther duty cycle, 
DC = 0 means output is low at all times and 1 means output is high at all times.
The delay input can delay a signal up to PT, this can be useful to synchronize different generators and generate interleaving signals.
in addition to a analog output Out there is a second boolean output Q.
*)
(* check dc = 1 or 0 *)
IF dc = 0 THEN
	out := am / -2 + os;
	Q := FALSE;
	RETURN;
ELSIF dc = 1 THEN
	out := am /2 + os;
	Q := TRUE;
	RETURN;
END_IF;

(* read system time and prepare input data *)
tx := TIME() - last;
DL := modR(dl,1);
IF dl < 0 THEN dl := 1 - dl; END_IF;
dc := modR(dc,1);
IF dc < 0 THEN dc := 1 - dc; END_IF;

(* init section *)
IF NOT init THEN
	init := TRUE;
	last := tx;
	tx := t#0s;
END_IF;

(* add last if one cycle is finished *)
IF tx >= pt THEN
	last := last + pt;
	tx := tx - pt;
END_IF;

(* check if falling or rising edge first *)
IF multime(pt, dl + dc) >= pt THEN
	(* generate falling edge *)
	IF tx >= multime(pt, dl + dc - 1) THEN
		out := am / -2 + os;
		Q := FALSE;
	END_IF;
	(* generate rising edge *)
	IF tx >= multime(pt, dl) THEN
		out := am / 2 + os;
		Q := TRUE;
	END_IF;
ELSE
	(* generate rising edge first *)
	IF tx >= multime(pt, dl) THEN
		out := am / 2 + os;
		Q := TRUE;
	END_IF;
	(* generate falling edge *)
	IF tx >= multime(pt, dl + dc) THEN
		out := am / -2 +os;
		Q := FALSE;
	END_IF;
END_IF;

(* revision history

hm	12. feb 2007		rev 1.1
	added default value for dc = 0.5

*)
END_FUNCTION_BLOCK

(* POU Heat_index, ST *)
FUNCTION Heat_index : REAL
VAR_INPUT
	T : REAL;
	RH : REAL;
END_VAR
VAR
	RH2 : REAL;
	T2 : REAL;
END_VAR

(*
version 1.1	27 Feb 2007
programmer 	hugo
tested by		tobias

this function calculates the heat index temperature depending on external temperature and Relative humidity

*)
IF RH < 20 OR T < 20 THEN
	Heat_index := T;
ELSE
	RH2 := EXPT(RH, 2);
	T := C_to_F(T);
	T2 := EXPT(T, 2);
	Heat_index := -42.379 + 2.04901523 * T + 10.1433127 * RH - 0.22475541 * T * RH - 6.83783E-3 * T2 - 5.481717E-2 * RH2
		+ 1.22874E-3 * T2 * RH + 8.5282E-4 * T * RH2 - 1.99E-6 * T2 * RH2;
	Heat_index := F_to_C(Heat_index);
END_IF;

(* revision history

hm 27.2.2007		rev 1.1
	deleted unused variables rh3 and T3
*)
END_FUNCTION

(* POU Heat_temp, ST *)
FUNCTION_BLOCK Heat_temp
VAR_INPUT
	T_ext : REAL;
	Offset : REAL;
	t_req : REAL;
END_VAR
VAR_INPUT CONSTANT
	TY_max : REAL := 70;
	TY_min : REAL := 20;
	T_int : REAL := 20;
	TY_config : REAL := 50;
	T_ext_config : REAL := -15;
	C : REAL := 1.33;
END_VAR
VAR_OUTPUT
	Ty : REAL;
END_VAR
VAR
END_VAR

(*
version 1.0	27 jan 2007
programmer 	hugo
tested by		tobias

Heat_Temp calculates a heat characteristic based on the formula: tv=ti+(tvmax-ti)*((ti-tau)/(ti-taumin))^(1/n)
while
tv necessary heating temperature.
ti internal room temperature (20°C)
tau current external temperature
external temperature to determine characteristics
C exponent for heating system (normally 1,33 or 1,1 for floor heating)

The two additional inputs TY_min and TY_max set limits for the output TY, while an offset inputs allows to rise or lower the room temperature.

*)
IF t_ext > t_int + Offset THEN
	ty := t_int + offset;
ELSE
Ty := T_int - offset + (TY_config - T_int) * EXPT((T_int - offset - T_ext) / (T_int - offset - T_ext_config),1 / C);
END_IF;
IF t_req > ty THEN ty := t_req; END_IF;
ty := LIMIT(TY_min, ty, TY_max);



(*

tv=ti+(tvmax-ti)*((ti-tau)/(ti-taumin))^(1/n)

tv aktuelle Vorlauftemp.
ti Raumtemperatur innen (20°C)
tau aktuelle Außentemperatur
taumin minimale Außentemperatur -12°C oder -15°C
n Heizkörperexponent (meistens 1,33)
Fußbodenheizung = 1,1
Wandheizung 1,3

Normen z. B. DIN 4703, DIN 4725 oder die Literatur, z. B Recknagel Abschnitt 1.3.5.

*)
END_FUNCTION_BLOCK

(* POU holiday, ST *)
FUNCTION_BLOCK holiday
VAR_INPUT
	date_in : DATE;
END_VAR
VAR CONSTANT
	size : INT := 24;
	feiertag : ARRAY [0..24] OF STRING(27) := 'Neujahr', 'Heilig Drei Könige', 'Karfreitag', 'Ostersonntag', 'Ostermontag', 'Tag der Arbeit',
	'Christi Himmelfahrt', 'Pfingstsonntag', 'Pfingstmontag', 'Fronleichnam', 'Augsburger Friedensfest', 'Maria Himmelfahrt',
	'Tag der Deutschen Einheit', 'Reformationstag', 'Allerheiligen', 'Buss und Bettag', '1. Weihnachtstag', '2. Weihnachtstag';
	f_day : ARRAY [0..24] OF SINT := 1, 6, -2, 0, 1, 1, 39, 49, 50 , 60, 8, 15, 3, 31, 1, 23, 25, 26;
	f_month : ARRAY [0..24] OF SINT := 1, 1, 0, 0, 0, 5, 0, 0, 0, 0, 8, 8, 10, 10, 11, 11, 12, 12;
	(* if month = 0 then F_day is the offset in days from easter *)
	f_use : ARRAY [0..24] OF SINT := 1,1,1,1,1,1,1,1,1,1,0,1,1,0,1,-3,1,1;
	(* 0 = not used, 1 = used, -1..-7 menas the weekday before the specified date example -3 means wednesday before 23.11 *)
END_VAR
VAR_OUTPUT
	Y : BOOL;
	name : STRING(20);
END_VAR
VAR
	last_active : DATE;
	ostern: DATE;
	i: INT;
	jahr: INT;
	x_date: DATE;
END_VAR

(*
version 1.1	28 feb 2007
programmer 	hugo
tested by		tobias

holiday calculates if a given day is a holiday and displays the name of the holiday as string as well as a boolean flag to indicate a holiday.
the holidays can be specified in an array in the constants section of the function block.
a holiday can be of fixed date for example new years day on january 1st.
a holiday can have a fixed offset from easter sunday as for most church holidays.
a holiday can be a specific weekday before a fixed date, for example buss und bettag is the last wednesday before nov 23rd.
with a simple f_use flag any specific holiday can be turned on or of if needed.

*)
(* for performance reasons only activate once a day *)
IF last_active = date_in THEN RETURN; END_IF;

(* berechnung von ostern für das aktuelle jahr *)
jahr := year(date_in);
Ostern := easter(jahr);
last_active := Date_in;

(* check array if today is holiday *)
Y := 0;
name := '';
FOR i := 0 TO size DO
	x_date := set_Date(jahr, f_month[i], f_day[i]);
	IF f_use[i] = 1 AND f_month[i] > 0 THEN
		(* check for fixed date holiday *)
		IF x_date = date_in THEN
			Y := TRUE;
			name := feiertag[i];
			RETURN;
		END_IF;
	ELSIF f_use[i] = 1 AND f_month[i] = 0 THEN
		(* check for holiday in reference to easter *)
		IF date_add(ostern,f_day[i] ,0,0,0) = date_in THEN
			Y := TRUE;
			name := feiertag[i];
			RETURN;
		END_IF;
	ELSIF f_use[i] < 0 THEN
		(* check for holiday on a weekday before date *)
		IF weekday(date_in) = ABS(f_use[i]) AND date_in < x_date AND date_in >= date_add(x_date,-7,0,0,0) THEN
			Y := TRUE;
			name := feiertag[i];
			RETURN;
		END_IF;
	END_IF;
END_FOR;

(* revision history
hm 27.2.2007	rev 1.1
	deleted unused variable init
*)

(*
Neujahrstag 	1. Januar 	• 	• 	• 	• 	• 	• 	• 	• 	• 	• 	• 	• 	• 	• 	• 	•
Heilige Drei Könige 	6. Januar 	• 	• 												• 		
Karfreitag 	Ostersonntag - 2d 	• 	• 	• 	• 	• 	• 	• 	• 	• 	• 	• 	• 	• 	• 	• 	•
Ostersonntag 	siehe Osterdatum 				(•) 												
Ostermontag 	Ostersonntag + 1d 	• 	• 	• 	• 	• 	• 	• 	• 	• 	• 	• 	• 	• 	• 	• 	•
Tag der Arbeit 	1. Mai 	• 	• 	• 	• 	• 	• 	• 	• 	• 	• 	• 	• 	• 	• 	• 	•
Christi Himmelfahrt 	Ostersonntag + 39d 	• 	• 	• 	• 	• 	• 	• 	• 	• 	• 	• 	• 	• 	• 	• 	•
Pfingstsonntag 	Ostersonntag + 49d 				(•) 												
Pfingstmontag 	Ostersonntag + 50d 	• 	• 	• 	• 	• 	• 	• 	• 	• 	• 	• 	• 	• 	• 	• 	•
Fronleichnam 	Ostersonntag + 60d 	• 	• 					• 			• 	• 	• 	1) 			2)
Augsburger Friedensfest 	8. August 		(3) 														
Mariä Himmelfahrt 	15. August 		(5) 										• 				
Tag der Deutschen Einheit 	3. Oktober 6) 	• 	• 	• 	• 	• 	• 	• 	• 	• 	• 	• 	• 	• 	• 	• 	•
Reformationstag 	31. Oktober 				• 				• 					• 	• 		•
Allerheiligen 	1. November 	• 	• 								• 	• 	• 				
Buß- und Bettag 4) 	Mittwoch vor dem 23.11. 			7 										• 			
1. Weihnachtstag 	25. Dezember 	• 	• 	• 	• 	• 	• 	• 	• 	• 	• 	• 	• 	• 	• 	• 	•
2. Weihnachtstag 	26. Dezember 	• 	• 	• 	• 	• 	• 	• 	• 	• 	• 	• 	• 	• 	• 	• 	•
*)
END_FUNCTION_BLOCK

(* POU hour_to_time, ST *)
FUNCTION hour_to_time : TIME
VAR_INPUT
	input : REAL;
END_VAR
VAR
END_VAR

(*
version 1.0	4 aug 2006
programmer 	hugo
tested by		tobias

converts an amount of hours in real to time
execution TIME on wago 750-841 =  17us
*)
hour_to_time := DWORD_TO_TIME(REAL_TO_DWORD(input * 3600000));
END_FUNCTION

(* POU hour_to_tod, ST *)
FUNCTION hour_to_tod : TOD
VAR_INPUT
	input : REAL;
END_VAR
VAR
END_VAR

(*
version 1.0	4 aug 2006
programmer 	hugo
tested by		tobias

converts an amount of hours in real to time of day 
execution time on wago 750-841 =  17us 
*)
hour_to_tod := DWORD_TO_TOD(REAL_TO_DWORD(input * 3600000));
END_FUNCTION

(* POU hyst_1, ST *)
FUNCTION_BLOCK hyst_1
VAR_INPUT
	In : REAL;
	high : REAL;
	low : REAL;
END_VAR
VAR_OUTPUT
	Q : BOOL := 0;
	win : BOOL := 0;
END_VAR
VAR
END_VAR

(*
	version 1.0	4 aug 2006
	programmer 	hugo
	tested BY		tobias

this hysteresis function switches the output high if the input signal reaches obove high and will switch to low when the input falls back below low value.
a separate output mid is set if the input stays between low and high value.

*)
IF Q THEN
	IF in < low THEN q := FALSE; END_IF;
ELSE
	IF in > high THEN q := TRUE; END_IF;
END_IF;
win := in > low AND in < high;
END_FUNCTION_BLOCK

(* POU hyst_2, ST *)
FUNCTION_BLOCK hyst_2
VAR_INPUT
	In : REAL;
	val : REAL;
	hys : REAL;
END_VAR
VAR_OUTPUT
	Q : BOOL := 0;
	win: BOOL;
END_VAR
VAR
	X : REAL;
END_VAR


(*
	version 1.0	4 aug 2006
	programmer 	oscat
	tested BY		tobias

this hysteresis function switches the output high if the input signal reaches obove val + hys/2 and will switch to low when the input falls back below val - hys/2 value.
a separate output mid is set if the input stays between low and high value.

*)
X := hys / 2;
IF Q THEN
	IF in < val - x THEN q := FALSE; END_IF;
ELSE
	IF in > val + x THEN q := TRUE; END_IF;
END_IF;
win := in > val - x AND in < val + x;
END_FUNCTION_BLOCK

(* POU Hyst_3, ST *)
FUNCTION_BLOCK Hyst_3
VAR_INPUT
	in : REAL;
	hyst : REAL;
	val1 : REAL;
	val2 : REAL;
END_VAR
VAR_OUTPUT
	Q1 : BOOL;
	Q2 : BOOL;
END_VAR
VAR
END_VAR

(*
	version 1.0	22 jan 2007
	programmer 	oscat
	tested BY		tobias

this is a double hysteresis function. Out1 follows a hysteresis function defined by val1and hyst, while out 2 follows val2 and hyst.
if the input signal is between the two hysteresis switches (val1 and val2) then non of the outputs is active.

*)
IF in < val1 - hyst / 2 THEN
	q1 := TRUE;
ELSIF in > val1 + hyst /2 THEN
	q1 := FALSE;
END_IF;
IF in < val2 - hyst / 2 THEN
	q2 := FALSE;
ELSIF in > val2 + hyst / 2 THEN
	q2 := TRUE;
END_IF;
END_FUNCTION_BLOCK

(* POU inc, ST *)
FUNCTION inc : INT
VAR_INPUT
	X : INT;
	D : INT;
	M : INT;
END_VAR
VAR
END_VAR


(*
version 1.0	7 feb 2007
programmer 	hugo
tested by		tobias

This is a increment function which increments the input X by the value D and compares the result with M.
if the output exceeds M it will continue to count from 0 again.

*)
inc := (X + D) MOD (m+1);
END_FUNCTION

(* POU inc_dec, ST *)
FUNCTION_BLOCK inc_dec
VAR_INPUT
	CHa : BOOL;
	CHb : BOOL;
	RST : BOOL := 0;
END_VAR
VAR_OUTPUT
	dir : BOOL;
	cnt : INT;
END_VAR
VAR
	edgea : BOOL := 0;
	clk: BOOL;
	clka: BOOL;
	clkb: BOOL;
	edgeb: BOOL;
	axb: BOOL;
END_VAR

(*
	version 1.0	4 aug 2006
	programmer 	oscat
	tested BY		oscat

incremental decoder with quadruple accuracy.
2 pulses for each channel are created for each directional pulse.
*)
axb := cha XOR chb;

(* create pulses for channel a *)
clka := cha XOR edgea;
edgea := cha;

clkb := chb XOR edgeb;
edgeb := chb;

(* create pulses for both channels *)
clk := clka OR clkb;

(* set the direction output *)
IF axb AND clka THEN dir := TRUE; END_IF;
IF axb AND clkb THEN dir := FALSE; END_IF;

(* increment or decrement the counter *)
IF clk AND dir THEN cnt := cnt + 1; END_IF;
IF clk AND NOT dir THEN cnt := cnt -1; END_IF;

(* reset the counter if rst active *)
IF rst THEN cnt := 0; END_IF;
END_FUNCTION_BLOCK

(* POU K_to_C, ST *)
FUNCTION K_to_C : REAL
VAR_INPUT
	Kelvin : REAL;
END_VAR
VAR
END_VAR

(*
version 1.0	4 dec 2006
programmer 	hugo
tested by		tobias

this function converts kelvin to celsius
*)
K_to_C := Kelvin + 273.15;
END_FUNCTION

(* POU KMH_TO_MS, ST *)
FUNCTION KMH_TO_MS : REAL
VAR_INPUT
	kmh : REAL;
END_VAR
VAR
END_VAR

(*
version 1.0	4 Feb 2007
programmer 	hugo
tested by		tobias

this function converts velocities from Kilometers / hour to Meters / Second

*)
KMH_TO_MS := kmh / 3.6;
END_FUNCTION

(* POU leap_of_Date, ST *)
FUNCTION leap_of_Date : BOOL
VAR_INPUT
	idate : DATE;
END_VAR
VAR
END_VAR

(*
version 1.1	2 oct 2006
programmer 	hugo
tested by		tobias


leap_year is true if the tested year is a leap year  
execution time on wago 750-841 =  30 us   
*)
leap_of_Date := leap_year(year(idate));


(* change history

2.10.2006		changes to rev 1.1
the function now calls leap_year to accomodate further accuracy.
the function now works for any year from 1970 to 2100

*)
END_FUNCTION

(* POU leap_year, ST *)
FUNCTION leap_year : BOOL
VAR_INPUT
	yr : INT;
END_VAR
VAR
END_VAR

(*
version 1.1	2 oct 2006
programmer 	hugo
tested by		tobias


leap_year is true if the tested year is a leap year  
execution time on wago 750-841 =  12 us    
*)
IF yr MOD 400 = 0 THEN leap_year := TRUE;
ELSIF yr MOD 100 = 0 THEN leap_year := FALSE;
ELSIF yr MOD 4 =0 THEN leap_year := TRUE;
ELSE leap_year := FALSE;
END_IF;


(* change history

2.10.2006		changes to rev 1.1
the function now works for any year from 1970 up to 2100

*)
END_FUNCTION

(* POU legionella, ST *)
FUNCTION_BLOCK legionella
VAR_INPUT
	manual : BOOL;
	temp_boiler : REAL;
	temp_return : REAL := 100;
	DT_in: DT;
	rst : BOOL;
END_VAR
VAR_INPUT CONSTANT
	T_start: TOD := tod#03:00:00;
	day : INT := 7;
	temp_set : REAL := 70;
	temp_offset : REAL := 10;
	temp_hys : REAL := 5;
	t_max_heat: TIME := t#10m;
	t_max_ret : TIME := t#10m;
	tp_0: TIME := t#5m;
	tp_1: TIME := t#5m;
	tp_2: TIME := t#5m;
	tp_3: TIME := t#5m;
	tp_4: TIME := t#5m;
	tp_5: TIME := t#5m;
	tp_6: TIME := t#5m;
	tp_7: TIME := t#5m;
END_VAR
VAR_OUTPUT
	Heat : BOOL;
	pump : BOOL;
	valve0 : BOOL;
	valve1 : BOOL;
	valve2 : BOOL;
	valve3 : BOOL;
	valve4 : BOOL;
	valve5 : BOOL;
	valve6 : BOOL;
	valve7 : BOOL;
	run: BOOL;
	Status : BYTE;
END_VAR
VAR
	X1: timer_1;
	x2: sequence_8;
	x3: hyst_1;
	init: BOOL;
END_VAR

(*
version 1.1	17. jan 2007
programmer 	oscat
tested by		hans

Legionella is a complete sequencer for up to 8 hot water lines that need to be sterilzed periodically.
legionella needs a DT input with the appropriate time, usually gererated by the rtc of the system. for system independence this time is connected externally.
T_start is the time when sterilazation should be started and day is the day_of_week when it should be performed (1=Monday and 7=sunday).
so sterilazation is autioimatically performed once a week at a specified time.
temp_set and temp_hys and temp_offset specify the boiler temperatur nedded for sterilization. as a defaut Temp_set is set to 70 deg C and Temp_hys is set to 5 deg C and temp_offset is 10 deg C.
a temp boiler input reads the boiler temperature of the hot water tank.
after a start pulse is gererated by the weekly timer or a manual test input the sequence is started:
1. the boiler is heated to temp_set + temp_offset + temp_hys = 85 deg C unless chaged at setup.
	the heat output is turned on and tells the heater to turn heating on. if the temp is not reached for a time of t_max_heat (10 min) the error output is set and the sequence is stopped.
2. after the specified temperature is reached, the output valve0 and pump is turned on and starts sterilization of line0 until temp_return has reached temp_set and continues to sterilize for a time of tp_0 (5 min default).
	if tmep_set is not reached at the temp_return_input then the error output is set and the sequence will be stopped.
	if there is no temp sensor for temp_return (the temperature at the return point for the circulation pump pls set this imput to a value greater then temp_set (by default use 100 deg C).
	in this case sterilization is performed for the default times without monitoring the return temp.
3. this sequence is repeated for up to valves.

connection scheme:

temp_boiler:	input oif the boiler temperature sensor.
temp_hys:		config value for the heater hysteresis, preset to 5 deg C.
temp_offset:	config value for the heater temp_offset against temp_set, preset to 10 deg C.
temp_set:		config value for the specified sterilization temperature, preset to 70 deg C.
temp_return:	input of the circulation return line temperature sensor, if not availabe set this value to 100 deg C.
manual:		manual input to start the sterilization by hand for diagnostic purposes, rising edge active, leave low for automatic operation.
DT_in:			date,time input supplied by a external real time clock.
T_start:		time of day when the sterilization should be started.
day:			config value for day of week when the process should be started, preset to sunday.
t_max_hest:	tmax time to be needed for the heater to heat the hot water tank to the specified value, preset to 10 min.

*)
(* startup initialization *)
IF NOT init THEN
	init := TRUE;
	X1.start_day := day;
	X1.start_time := T_start;
	X3.low := Temp_offset + temp_set;
	X3.high := Temp_hys + X3.low;
	X2.wait0 := T_max_heat;
	X2.delay0 := TP_0;
	X2.delay1 := TP_1;
	X2.delay2 := TP_2;
	X2.delay3 := TP_3;
	X2.delay4 := TP_4;
	X2.delay5 := TP_5;
	X2.delay6 := TP_6;
	X2.delay7 := TP_7;
	X2.wait1 := T_max_ret;
	X2.wait2 := T_max_ret;
	X2.wait3 := T_max_ret;
	X2.wait4 := T_max_ret;
	X2.wait5 := T_max_ret;
	X2.wait6 := T_max_ret;
	X2.wait7 := T_max_ret;
	X2();
END_IF;

(* oerational code *)
X1(DT_in := DT_in);
IF X1.Q OR manual OR x2.run THEN
	X3(in := temp_boiler);
	X2.in0 := X3.Q OR x3.win;
	X2.in1 := temp_return >= temp_set;
	X2.in2 := x2.in1;
	X2.in3 := x2.in1;
	X2.in4 := x2.in1;
	X2.in5 := x2.in1;
	X2.in6 := x2.in1;
	X2.in7 := x2.in1;
	X2.rst := rst;
	X2(start := X1.Q OR manual);
	run := x2.run;
	pump := x2.any;
	Heat := NOT X3.Q AND x2.run;
	valve0 := X2.Q0;
	valve1 := X2.Q1;
	valve2 := X2.Q2;
	valve3 := X2.Q3;
	valve4 := X2.Q4;
	valve5 := X2.Q5;
	valve6 := X2.Q6;
	valve7 := X2.Q7;
	pump := X2.any;
	status := X2.status;
ELSE;
	X2(start :=0);
	status := x2.status;
END_IF;

(* revision history

hm 17.jan 2007	rev 1.1
	rewritten to st for higher performance
	changes eeror output to esr compatible status output
*)
END_FUNCTION_BLOCK

(* POU timer_1, ST *)
FUNCTION_BLOCK timer_1
VAR_INPUT
	DT_in : DT;
	start_time : TOD;
	duration : TIME;
	start_day : INT := 0;
END_VAR
VAR_OUTPUT
	Q : BOOL;
END_VAR
VAR
	last_check : TIME := T#0s;
	last: DATE;
	dat: DATE;
END_VAR

(*
version 1.2	25 dec 2006
programmer 	oscat
tested by		tobias

this is a simple timer that generates an output pulse once a day if start_day = 0.
if start_day is a number from 1 .. 7 then a output pulse is generated for the respective weekday 1 = monday.
the output pulse width can be programmed, if set to 0 a pulse is generated for one cycle only.

*)
IF TIME() - last_check >= T#1s THEN
	dat := DT_TO_DATE(dt_in);
	IF NOT Q AND (start_day = 0 OR start_day = weekday(dat)) AND dat <> last AND DT_TO_TOD(dt_in) >= start_time THEN
		Q := TRUE;
		last := dat;
	ELSIF Q AND DT_TO_TOD(dt_in) >= start_time + duration THEN
		Q := FALSE;
	END_IF;
	last_check := TIME();
END_IF;

(*
1.12.2006 hm		rev 1.1
corrected an error with pulse width = 0.

25.12.2006 hm	rev 1.2
corrected an error when timeer overflows.

*)
END_FUNCTION_BLOCK

(* POU sequence_8, ST *)
FUNCTION_BLOCK sequence_8
VAR_INPUT
	in0 : BOOL := TRUE;
	in1 : BOOL := TRUE;
	in2 : BOOL := TRUE;
	in3 : BOOL := TRUE;
	in4 : BOOL := TRUE;
	in5 : BOOL := TRUE;
	in6 : BOOL := TRUE;
	in7 : BOOL := TRUE;
	start : BOOL;
	rst : BOOL;
	wait0 : TIME := t#0s;
	delay0 : TIME := t#0s;
	wait1 : TIME := t#0s;
	delay1 : TIME := t#0s;
	wait2 : TIME := t#0s;
	delay2 : TIME := t#0s;
	wait3 : TIME := t#0s;
	delay3 : TIME := t#0s;
	wait4 : TIME := t#0s;
	delay4 : TIME := t#0s;
	wait5 : TIME := t#0s;
	delay5 : TIME := t#0s;
	wait6 : TIME := t#0s;
	delay6 : TIME := t#0s;
	wait7 : TIME := t#0s;
	delay7 : TIME := t#0s;
END_VAR
VAR_INPUT CONSTANT
	stop_on_error : BOOL := FALSE;
END_VAR
VAR_OUTPUT
	Q0 : BOOL;
	Q1 : BOOL;
	Q2 : BOOL;
	Q3 : BOOL;
	Q4 : BOOL;
	Q5 : BOOL;
	Q6 : BOOL;
	Q7 : BOOL;
	any : BOOL;
	run: BOOL;
	step : INT := -1;
	status : BYTE;
END_VAR
VAR
	last : TIME;
	edge : BOOL;
	tx: TIME;
	init: BOOL;
END_VAR

(*
version 1.3	17 jan 2007
programmer 	oscat
tested by		hans

sequence_8 enables run when a low to high transition is present on start.
a low to high transition on start will restart the sequencer at any time while a rst will hold the sequencer in reset while true.
after run is enabled with a rising edge on start the sequencer waits for wait0 on in0 to enable q0 which stays on for delay0.
the next cycle starts with wait1, continues with delay 1 and so on...
if an edge is not detected during the wait period, the sequencer will then display the error number on the status output.
The status numbers are 1 .. 8 for erros in step 0..7.
after the last step that sets q7, the sequencer leaves q7 on for delay7 and then resets to the initial state.
a step output will indicate the current step of the sequencer and will also be present with a fault condition.
after the first output is turened on the sequencer switches from q0 to q1 and so on, at any time there is only one output enabled.
if an input signal is not detected during a wait period, the sequencer will display the error number ( 1 for in0, 2 for in1 .... ).
when an error is present and the config variable stop_on_error is set then the sequencer will stop. otherwise it will continue.
The status output will also display 110 for waiting and 111 sequece running.

*)
(* read sps timer *)
tx := TIME();

(* initialize on startup *)
IF NOT init THEN
	last := tx;
	init := TRUE;
	status := 110;
END_IF;

(* asynchronous reset *)
IF rst THEN
	step := -1;
	Q0 := 0;
	Q1 := 0;
	Q2 := 0;
	Q3 := 0;
	Q4 := 0;
	Q5 := 0;
	Q6 := 0;
	Q7 := 0;
	status := 110;
	run := 0;

(* edge on start input restarts the sequencer *)
ELSIF start AND NOT edge THEN
	step := 0;
	last := tx;
	status := 111;
	Q0 := 0;
	Q1 := 0;
	Q2 := 0;
	Q3 := 0;
	Q4 := 0;
	Q5 := 0;
	Q6 := 0;
	Q7 := 0;
	run := 1;
END_IF;
edge := start;

(* check if stop on error is necessary *)
IF status > 0 AND status < 100 AND stop_on_error THEN RETURN; END_IF;

(* sequence is running *)
IF run AND step = 0 THEN
	IF NOT q0 AND in0 AND tx - last <= wait0 THEN
		Q0 := TRUE;
		last := tx;
	ELSIF NOT q0 AND tx - last > wait0 THEN
		status := 1;
		run := FALSE;
	ELSIF q0 AND tx - last >= delay0 THEN
		step := 1;
		last := tx;
	END_IF;
END_IF;
IF run AND step = 1 THEN
	IF NOT q1 AND in1 AND tx - last <= wait1 THEN
		Q0 := FALSE;
		Q1 := TRUE;
		last := tx;
	ELSIF NOT q1 AND Tx - last > wait1 THEN
		status := 2;
		q0 := FALSE;
		run := FALSE;
	ELSIF q1 AND tx - last >= delay1 THEN
		step := 2;
		last := tx;
	END_IF;
END_IF;
IF run AND step = 2 THEN
	IF NOT q2 AND in2 AND tx - last <= wait2 THEN
		Q1 := FALSE;
		Q2 := TRUE;
		last := tx;
	ELSIF NOT q2 AND Tx - last > wait2 THEN
		status := 3;
		q1 := FALSE;
		run := FALSE;
	ELSIF q2 AND tx - last >= delay2 THEN
		step := 3;
		last := tx;
	END_IF;
END_IF;
IF run AND step = 3 THEN
	IF NOT q3 AND in3 AND tx - last <= wait3 THEN
		Q2 := FALSE;
		Q3 := TRUE;
		last := tx;
	ELSIF NOT q3 AND Tx - last > wait3 THEN
		status := 4;
		q2 := FALSE;
		run := FALSE;
	ELSIF q3 AND tx - last >= delay3 THEN
		step := 4;
		last := tx;
	END_IF;
END_IF;
IF run AND step = 4 THEN
	IF NOT q4 AND in4 AND tx - last <= wait4 THEN
		Q3 := FALSE;
		Q4 := TRUE;
		last := tx;
	ELSIF NOT q4 AND Tx - last > wait4 THEN
		status := 5;
		q3 := FALSE;
		run := FALSE;
	ELSIF q4 AND tx - last >= delay4 THEN
		step := 5;
		last := tx;
	END_IF;
END_IF;
IF run AND step = 5 THEN
	IF NOT q5 AND in5 AND tx - last <= wait5 THEN
		Q4 := FALSE;
		Q5 := TRUE;
		last := tx;
	ELSIF NOT q5 AND Tx - last > wait5 THEN
		status := 6;
		q4 := FALSE;
		run := FALSE;
	ELSIF q5 AND tx - last >= delay5 THEN
		step := 6;
		last := tx;
	END_IF;
END_IF;
IF run AND step = 6 THEN
	IF NOT q6 AND in6 AND tx - last <= wait6 THEN
		Q5 := FALSE;
		Q6 := TRUE;
		last := tx;
	ELSIF NOT q6 AND Tx - last > wait6 THEN
		status := 7;
		q5 := FALSE;
		run := FALSE;
	ELSIF q6 AND tx - last >= delay6 THEN
		step := 7;
		last := tx;
	END_IF;
END_IF;
IF run AND step = 7 THEN
	IF NOT q7 AND in7 AND tx - last <= wait7 THEN
		Q6 := FALSE;
		Q7 := TRUE;
		last := tx;
	ELSIF NOT q7 AND Tx - last > wait7 THEN
		status := 8;
		q6 := FALSE;
		run := FALSE;
	ELSIF q7 AND tx - last >= delay7 THEN
		step := -1;
		Q7 := FALSE;
		Run := FALSE;
		status := 110;
	END_IF;
END_IF;
any := q0 OR q1 OR q2 OR q3 OR q4 OR q5 OR q6 OR q7;

(*
hm 1.10.06		rev 1.1
	corrected delay logic to be after event and not before
	added any output

hm 1.12.06		rev 1.2
	corrected failure in sequence logic.
	added init at startup to prevent from initial statuss after start.

hm 17.1.2007		rev 1.3
	changed output fault to status for better compatibility with other modules (ESR)
	added stop on error functionality and setup variable
	default for inputs in0..7 is true.
	renames variable state to step
*)
END_FUNCTION_BLOCK

(* POU local_time, ST *)
FUNCTION local_time : DT
VAR_INPUT
	utc : DT;
	time_zone_offset : TIME;
	dst_enable: BOOL;
END_VAR
VAR
END_VAR

(*
version 1.1	2 oct 2006
programmer 	hugo
tested by		tobias

localtime calculates the local time according to DSTenable and time_zone_offset.
the dst input only tells the function the dst (daylight savings time) is enabled but the calculation for summertime on and off is done by the function itself.
this means the dst input only tells the function to switch summertime on and off automatically or not.
the function will switch to summertime automatically at the specified time end of march and back end of october.
the summertime calculation is done according to european standards.
the input is world time (UTC) and a given time_zone_offset for any time_zone.

execution time on wago 750-841 = 140 us   
*)
IF DST(utc,time_zone_offset) AND dst_enable THEN
	local_time := utc + time_zone_offset + T#1h;
ELSE
	local_time := utc + time_zone_offset;
END_IF;


(*

change history

2.10.2006 hm	rev 1.1
	corrected an error in the dst check for correct function

*)
END_FUNCTION

(* POU lowercase, ST *)
FUNCTION lowercase : STRING
VAR_INPUT
	str : STRING;
END_VAR
VAR
	PT : POINTER TO BYTE;
	pos: INT;
END_VAR

(*
version 1.0	6 oct 2006
programmer 	hugo
tested by		tobias

uppercase returns str while all letters A..Z are converted to lowercase.
*)
PT := ADR(lowercase);
lowercase := str;
FOR pos := 1 TO LEN(lowercase) DO
	IF PT^ > 64 AND PT^ < 91 THEN PT^ := PT^ + 32; END_IF;
	PT := PT + 1;
END_FOR;
END_FUNCTION

(* POU LTCH, ST *)
FUNCTION_BLOCK LTCH
VAR_INPUT
	D : BOOL;
	L : BOOL;
	RST : BOOL := 0;
END_VAR
VAR_OUTPUT
	Q : BOOL := 0;
END_VAR
VAR
END_VAR

(*
version 1.0	4 aug 2006
programmer 	hugo
tested by		tobias

Transparent Latch with asynchronous reset

executioin TIME on wago 750-841 = 5us
*)
(* as long as L is true, the latch is transparent and and change of D is transferred to Q *)
(* of course only when there is no asynchronous reset *)
IF L AND NOT rst THEN Q := D;	(* latch is transparent *)
ELSIF rst THEN Q:= 0;			(* if asynchronous reset then Q=0 *)
END_IF;
END_FUNCTION_BLOCK

(* POU LTCH_4, ST *)
FUNCTION_BLOCK LTCH_4
VAR_INPUT
	D0 : BOOL;
	D1 : BOOL;
	D2 : BOOL;
	D3 : BOOL;
	L : BOOL;
	RST : BOOL := 0;
END_VAR
VAR_OUTPUT
	Q0 : BOOL := 0;
	Q1 : BOOL := 0;
	Q2 : BOOL := 0;
	Q3 : BOOL := 0;
END_VAR
VAR
END_VAR

(*
version 1.0	4 aug 2006
programmer 	hugo
tested by		tobias

Quad Transparent Latch with asynchronous reset

executioin TIME on wago 750-841 = 5us
*)
(* as long as L is true, the latch is transparent and and change of D is transferred to Q *)
(* of course only when there is no asynchronous reset *)
IF L AND NOT rst THEN
	Q0 := D0;	(* latch is transparent *)
	Q1 := D1;
	Q2 := D2;
	Q3 := D3;
ELSIF rst THEN
	Q0 := FALSE;			(* if asynchronous reset then Q=0 *)
	Q1 := FALSE;
	Q2 := FALSE;
	Q3 := FALSE;
END_IF;
END_FUNCTION_BLOCK

(* POU Ltime, ST *)
FUNCTION_BLOCK Ltime
VAR_INPUT
	UTC : DT;
	dst_enable : BOOL;
	time_zone_offset : TIME;
END_VAR
VAR_OUTPUT
	local_DT : DT;
	DST_on : BOOL;
	wday : INT;
END_VAR
VAR
	time_adder : TIME := t#0s;
	next_check : DT := dt#1970-01-01-00:00:00;
END_VAR

(*

version 1.2	17 jan 2007
programmer 	oscat
tested by		tobias

ltime is a real time clock that uses the system rtc as utc time and calculates and given time zone.
the utc time is supplied on the input UTC.
according to the input variable time_zone_offset when the input dst_enable is true,
the dst on and off times are calculated by a formula for any given year and the time is advanced and reset by one hour
at 02:00 and 03:00 for the last sunday of march and last sunday of october.
the code is high performance and the rtc counts every second.
if more then one time zone is needed by the systen the clock can be started many times by placing more then one function block.

execution time on wago 750-841 = 20 us 
 
*)
IF local_dt > next_check THEN
	next_check := DWORD_TO_DT(DT_TO_DWORD(local_dt) / 3600 * 3600 +3600);
	dst_on := DST(local_dt,time_zone_offset);
	IF dst_on AND dst_enable THEN time_adder := time_zone_offset + T#1h; ELSE time_adder := time_zone_offset; END_IF;
END_IF;
local_dt :=utc + time_adder;
wday := weekday(DT_TO_DATE(local_dt));

(* revision history

hm 2.10.2006	rev 1.1
	corrected an error where dst would be delayed by 0.1second

hm 17.1.2007	rev 1.2
	added utc input instead of internal sysrtcgettime because this would only work on wago.
	dst_enable would not be checked before dst would be enabled.
*)
END_FUNCTION_BLOCK

(* POU m_t, ST *)
FUNCTION_BLOCK m_t
VAR_INPUT
	in: BOOL;
END_VAR
VAR_OUTPUT
	PT : TIME := t#0ms;
END_VAR
VAR
	edge : BOOL := 0;
	start: TIME;
	stop:TIME;
END_VAR

(*
	version 1.0	4 aug 2006
	programmer 	hugo
	tested BY		tobias

this measures the with of a pulse and returs the pulse width
*)
(* edge trigger rising and falling edge *)
IF in XOR edge THEN
	edge := in;
	(* rising edge starts measurement *)
	IF in THEN
		start := TIME();
	(* falling edge stops measurement *)
	ELSE
		stop := TIME();
		pt := stop - start;
	END_IF;
END_IF;
END_FUNCTION_BLOCK

(* POU m_tx, ST *)
FUNCTION_BLOCK m_tx
VAR_INPUT
	in: BOOL;
END_VAR
VAR_OUTPUT
	TH : TIME := t#0ms;
	TL : TIME := t#0ms;
	DC : REAL := 0;
	F: REAL;
END_VAR
VAR
	edge : BOOL := 0;
	start: TIME;
	stop:TIME;
END_VAR

(*
	version 1.0	4 aug 2006
	programmer 	oscat
	tested BY		oscat

this measures the timing of a signal
TH is the high ulse width
TL is the low pulse width
DC is the duty cycle
F is the frequency
the acuracy depends on the cycle time of the sps and is limited to 1ms resolution

*)
(* edge trigger rising and falling edge *)
IF in XOR edge THEN
	edge := in;
	(* rising edge starts measurement *)
	IF in THEN
		start := TIME();
		tl := start - stop;
		IF th > t#0ms THEN
			dc := TIME_TO_REAL(th) / TIME_TO_REAL(th+tl);
			f := 1000 / TIME_TO_REAL(th + tl);
		END_IF;
	(* falling edge starts second cycle measurement *)
	ELSE
		stop := TIME();
		th := stop - start;
		IF th > t#0ms THEN dc := TIME_TO_REAL(th) /  TIME_TO_REAL(th+tl);
			f := 1000 / TIME_TO_REAL(th + tl);
		END_IF;
	END_IF;
END_IF;
END_FUNCTION_BLOCK

(* POU max3, ST *)
FUNCTION max3 : REAL
VAR_INPUT
	in1 : REAL;
	in2 : REAL;
	in3 : REAL;
END_VAR
VAR
END_VAR

(*
version 1.0	1 jan 2007
programmer 	hugo
tested by		tobias

this function returns the highest of 3 real values

*)
IF in1 >= in2 AND in1 >= in3 THEN
	max3 := in1;
ELSIF in2 >= in1 AND in2 >= in3 THEN
	max3 := in2;
ELSE
	max3 := in3;
END_IF;
END_FUNCTION

(* POU mid3, ST *)
FUNCTION mid3 : REAL
VAR_INPUT
	in1 : REAL;
	in2 : REAL;
	in3 : REAL;
END_VAR
VAR
END_VAR

(*
version 1.1	1 jan 2007
programmer 	hugo
tested by		tobias

returns the mid value of 3 real inputs.

*)
IF (in1 <= in2) AND (in1 >= in3) OR (in1 >= in2) AND (in1 <= in3) THEN
	mid3 := in1;
ELSIF (in2 <= in1) AND (in2 >= in3) OR (in2 >= in1) AND (in2 <= in3) THEN
	mid3 := in2;
ELSE
	mid3 := in3;
END_IF;

(*
hm	1.1.2007	rev 1.1
	rewrote the function for better performance

*)
END_FUNCTION

(* POU min3, ST *)
FUNCTION min3 : REAL
VAR_INPUT
	in1 : REAL;
	in2 : REAL;
	in3 : REAL;
END_VAR
VAR
END_VAR

(*
version 1.0	1 jan 2007
programmer 	hugo
tested by		tobias

this function returns the lowest of 3 real values

*)
IF in1 <= in2 AND in1 <= in3 THEN
	min3 := in1;
ELSIF in2 <= in1 AND in2 <= in3 THEN
	min3 := in2;
ELSE
	min3 := in3;
END_IF;
END_FUNCTION

(* POU minute_to_time, ST *)
FUNCTION minute_to_time : TIME
VAR_INPUT
	input : REAL;
END_VAR
VAR
END_VAR

(*
version 1.0	4 aug 2006
programmer 	hugo
tested by		tobias

converts an amount of minutes in real to time
execution time on wago 750-841 =  17us
*) 
minute_to_time := DWORD_TO_TIME(REAL_TO_DWORD(input * 60000));
END_FUNCTION

(* POU MS_TO_KMH, ST *)
FUNCTION MS_TO_KMH : REAL
VAR_INPUT
	ms : REAL;
END_VAR
VAR
END_VAR

(*
version 1.0	4 Feb 2007
programmer 	hugo
tested by		tobias

this function converts velocities from Meters / Second to Kilometers / hour.

*)
MS_TO_KMH := ms * 3.6;
END_FUNCTION

(* POU MUL_ADD, ST *)
FUNCTION MUL_ADD : REAL
VAR_INPUT
	X : REAL;
	K : REAL := 1;
	O : REAL := 0;
END_VAR
VAR
END_VAR

(*
version 1.0	28 Feb 2007
programmer 	hugo
tested by		tobias

this function multiplies an input X with K and adds Offset O to the result.

*)
MUL_ADD := X * K + O;
END_FUNCTION

(* POU multi_in, ST *)
FUNCTION multi_in : REAL
VAR_INPUT
	in_1 : REAL;
	in_2 : REAL;
	in_3 : REAL;
	default : REAL;
	in_min : REAL;
	in_max : REAL;
	mode : BYTE;
END_VAR
VAR
	count: INT;
	F1: BOOL;
	F2: BOOL;
	F3: BOOL;
END_VAR

(*

version 1.1	1 jan 2007
programmer 	oscat
tested by		hugo

multi_in is a signal conditioning function ehich can be configured in 8 different ways.
it is used to read multiple sensors for the same value and protect the user from broken sensors or invalid data from sensors.

multi_in can be configured in different ways:
	mode = 0 means the the avg of the 3 inputs is used, this mode is the default mode.
	mode = 1 means in_1 is used.
	mode = 2 means in_2 is used.
	mode = 3 means in_3 is used.
	mode = 4 means default is used.
	mode = 5 means the lowest of the 3 external temperatures is used.
	mode = 6 means the higest externnal temperature is used.
	mode = 7 means the midlle input is used, if there are only two working, the lowest input is used.
	mode > 7 ,eans output is 0 at all times.
	in any config mode, an input higher then in_max or lower then in_min is ignored to prevent values from broken sensors or wires.
	if all inputs are higher then in_max or lower then in_min, a default value (default) is used.
*)
IF  in_1 > in_min AND in_1 < in_max THEN F1 := TRUE; ELSE F1 := FALSE; END_IF;
IF  in_2 > in_min AND in_2 < in_max THEN F2 := TRUE; ELSE F2 := FALSE; END_IF;
IF  in_2 > in_min AND in_3 < in_max THEN F3 := TRUE; ELSE F3 := FALSE; END_IF;

CASE mode OF
0:	count := 0;
	IF F1 THEN
		count := count + 1;
		multi_in := in_1;
	ELSE
		multi_in := 0;
	END_IF;
	IF F2 THEN
		count := count + 1;
		multi_in := multi_in + in_2;
	END_IF;
	IF F3 THEN
		count := count + 1;
		multi_in := multi_in + in_3;
	END_IF;
	IF count = 0 THEN
		multi_in := default;
	ELSE
		multi_in := multi_in / count;
	END_IF;

1:	IF F1 THEN multi_in := in_1; ELSE multi_in := default; END_IF;

2:	IF F2 THEN multi_in := in_2; ELSE multi_in := default; END_IF;

3:	IF F3 THEN multi_in := in_3; ELSE multi_in := default; END_IF;

4:	multi_in := default;

5:	IF F1 THEN multi_in := in_1; ELSE multi_in := in_max; END_IF;
	IF F2 AND in_2 < multi_in THEN multi_in := in_2; END_IF;
	IF F3 AND in_3 < multi_in THEN multi_in := in_3; END_IF;
	IF multi_in = in_max THEN multi_in := default; END_IF;

6:	IF F1 THEN multi_in := in_1; ELSE multi_in := in_min; END_IF;
	IF F2 AND in_2 > multi_in THEN multi_in := in_2; END_IF;
	IF F3 AND in_3 > multi_in THEN multi_in := in_3; END_IF;
	IF multi_in = in_min THEN multi_in := default; END_IF;

7:	IF F1 AND F2 AND F3 THEN multi_in := mid3(in_1, in_2, in_3);
	ELSIF F1 AND F2 THEN multi_in := MIN(in_1, in_2);
	ELSIF F1 AND F3 THEN multi_in := MIN(in_1, in_3);
	ELSIF F2 AND F3 THEN multi_in := MIN(in_2, in_3);
	ELSIF F1 THEN multi_in := in_1;
	ELSIF F2 THEN multi_in := in_2;
	ELSIF F3 THEN multi_in := in_3;
	ELSE multi_in := default;
	END_IF;

END_CASE;

(*
hm 1.1.2007	rev 1.1
	changed midr to mid3 function

*)
END_FUNCTION

(* POU mux_2, ST *)
FUNCTION mux_2 : BOOL
VAR_INPUT
	D0: BOOL;
	D1: BOOL;
	A0: BOOL;
END_VAR
VAR
END_VAR

(*
	version 1.1	5 oct 2006
	programmer 	hugo
	tested BY		tobias

	dual input multiplexer
	depending on the value of A0, D0 or D1 will be switched to the Output

	executioin TIME on wago 750-841 = 7us
*)
mux_2 := (D0 AND NOT A0) OR (D1 AND A0);

(*

change history:
5.10.2006		changed to ST Langage for better protability.

*)
END_FUNCTION

(* POU mux_4, ST *)
FUNCTION mux_4 : BOOL
VAR_INPUT
	D0: BOOL;
	D1: BOOL;
	D2: BOOL;
	D3: BOOL;
	A0: BOOL;
	A1: BOOL;
END_VAR
VAR
END_VAR

(*
	version 1.0	4 aug 2006
	programmer 	hugo
	tested BY		tobias

	quad input multiplexer
	depending on the value of A0 and A1, one of the 4 inputs will be switched to the Output

	executioin TIME on wago 750-841 = 13us
*)
mux_4 := (D0 AND NOT A0 AND NOT A1)
	OR (D1 AND A0 AND NOT A1)
	OR (D2 AND NOT A0 AND A1)
	OR (D3 AND A0 AND A1);


(* change history:

5.10.2006		rewritten to ST for better portability


*)
END_FUNCTION

(* POU MUX_R2, ST *)
FUNCTION MUX_R2 : REAL
VAR_INPUT
	IN0 : REAL;
	IN1 : REAL;
	A : BOOL;
END_VAR
VAR
END_VAR

(*
version 1.0	19 jan 2007
programmer 	oscat
tested by		tobias

MUX_R2 is an analog Multiplexer.
one of 2 real inputs are selected and put through to out.
The Adress input A selects between 2 Real inputs IN0 and IN1, A=0 > In0, A=1 > in1.

*)
IF NOT A THEN
	MUX_R2 := IN0;
ELSE
	MUX_R2 := IN1;
END_IF;
END_FUNCTION

(* POU MUX_R4, ST *)
FUNCTION MUX_R4 : REAL
VAR_INPUT
	IN0 : REAL;
	IN1 : REAL;
	IN2 : REAL;
	IN3 : REAL;
	A0 : BOOL;
	A1 : BOOL;
END_VAR
VAR
END_VAR

(*
version 1.0	19 jan 2007
programmer 	oscat
tested by		tobias

MUX_R4 is an analog Multiplexer.
one of 4 real inputs are selected and put through to out.
The Adress input A0 and A1 selects between the 4 Real inputs IN0.. IN1.

*)
IF NOT A0 AND NOT A1 THEN
	MUX_R4 := IN0;
ELSIF A0 AND NOT a1 THEN
	MUX_R4 := IN1;
ELSIF NOT A0 AND A1 THEN
	MUX_R4 := IN2;
ELSE
	MUX_R4 := IN3;
END_IF;
END_FUNCTION

(* POU Offset2, ST *)
FUNCTION Offset2 : REAL
VAR_INPUT
	X : REAL;
	O1, O2, O3, O4 : BOOL;
	D : BOOL;
END_VAR
VAR_INPUT CONSTANT
	Offset_1 : REAL;
	Offset_2 : REAL;
	Offset_3 : REAL;
	Offset_4 : REAL;
	default : REAL;
END_VAR

(*
version 1.0	12 jan 2007
programmer 	oscat
tested by		tobias

The Function offset adds offsets to an analog signal depending on digital inputs.
one offset can be added at the same time, if more then one input is true, the one with the highest number (o1 .. o4) will be used.
The input D will select a default value instead of X for input.

*) 
IF D THEN Offset2 := default; ELSE Offset2 := X; END_IF;
IF O4 THEN Offset2 := Offset2 + offset_4;
ELSIF O3 THEN Offset2 := Offset2 + offset_3;
ELSIF O2 THEN Offset2 := Offset2 + offset_2;
ELSIF O1 THEN Offset2 := Offset2 + offset_1;
END_IF;
END_FUNCTION

(* POU OM_to_F, ST *)
FUNCTION OM_to_F : REAL
VAR_INPUT
	OM : REAL;
END_VAR
VAR
END_VAR

(*
version 1.0	22 jan 2007
programmer 	hugo
tested by		tobias

this function converts Omega F to frequency
F = OM / (2*PI)
*)
OM_to_F := OM / PI2;
END_FUNCTION

(* POU Oscat_version, ST *)
FUNCTION Oscat_version : DWORD
VAR_INPUT
END_VAR
VAR
END_VAR


(*
version 1.0	6 oct 2006
programmer 	hugo
tested by		tobias

oscat_version returns the version number in dword format
132 is library version 1.32

*)
Oscat_version := 151;
END_FUNCTION

(* POU parity, ST *)
FUNCTION parity : BOOL
VAR_INPUT
	in : DWORD;
END_VAR
VAR
	i : INT;
	cnt : INT := 0;
END_VAR

(*
	version 1.0	1 sep 2006
	programmer 	hugo
	tested BY		hans

this function calculates the even parity of an input Dword
the output will be true if the amount of high bits are an odd number.

*)
FOR i := 0 TO 31 DO
	IF in.0 THEN cnt := cnt +1; END_IF;
	in := SHR(in,1);
END_FOR;
IF (cnt MOD 2) = 1 THEN parity := TRUE; ELSE parity := FALSE; END_IF;
END_FUNCTION

(* POU PT_to_F, ST *)
FUNCTION PT_to_F : REAL
VAR_INPUT
	PT : TIME;
END_VAR
VAR
END_VAR

(*
version 1.0	4 aug 2006
programmer 	hugo
tested by		tobias

this function converts periode time to frequency
*)
PT_to_F := 1000/DWORD_TO_REAL(TIME_TO_DWORD(PT));
END_FUNCTION

(* POU Pulse_Length, ST *)
FUNCTION_BLOCK Pulse_Length
VAR_INPUT
	in : BOOL;
END_VAR
VAR_OUTPUT
	short : BOOL;
	middle : BOOL;
	long : BOOL;
END_VAR
VAR_INPUT CONSTANT
	T_short : TIME := t#100ms;
	T_long : TIME := t#1s;
END_VAR
VAR
	tx : TIME;
	tn: TIME;
	edge : BOOL;
END_VAR

(*
version 1.0	15 Feb 2006
programmer 	oscat
tested by		tobias

*)
(* read system time *)
tx := TIME();

(* reset outputs, they should only be active 1 cycle *)
short := FALSE;
Middle := FALSE;
long := FALSE;

(* detect rising edge *)
IF in AND NOT edge THEN
	edge := TRUE;
	tn := tx;

(* detect for falling edge *)
ELSIF NOT in AND edge THEN
	edge := FALSE;
	tn := tx - tn;
	IF tn < t_short THEN
		short := TRUE;
	ELSIF tn > t_long THEN
		long := TRUE;
	ELSE
		Middle := TRUE;
	END_IF;

(* generate long pulse as soon as T_long is reached *)
ELSIF in AND tx - tn > t_long THEN
	long := TRUE;
END_IF;
END_FUNCTION_BLOCK

(* POU pwm_dc, ST *)
FUNCTION_BLOCK pwm_dc
VAR_INPUT
	F : REAL;
	DC : REAL;
END_VAR
VAR_OUTPUT
	Q : BOOL;
END_VAR
VAR
	clk: CLK_Prg;
	pulse: TP_R;
END_VAR

(*
	version 1.1	25 feb 2007
	programmer 	oscat
	tested BY		oscat

this signal generator generates a square wave signal which is specified by the frequency and the duty cycle
*)
CLK(PT := REAL_TO_TIME(1000/F));
Pulse(in := clk.Q, pt := REAL_TO_TIME(1000/F*DC));
Q := pulse.Q;

(* revision history

hm		25. feb 2007	rev 1.1
	recoded in st for better performance and better portability

*)
END_FUNCTION_BLOCK

(* POU TP_R, ST *)
FUNCTION_BLOCK TP_R
VAR_INPUT
	in : BOOL;
	PT : TIME;
END_VAR
VAR_OUTPUT
	Q : BOOL := 0;
	ET : TIME := t#0ms;
END_VAR
VAR
	edge : BOOL := FALSE;
	start : TIME := t#0ms;
END_VAR

(*
version 1.0	4 aug 2006
programmer 	hugo
tested by		tobias

retriggerable edge triggered pulse similar to TP but with a retrigger function
if the pt input is 0 then output is always low.
*)
(* rising edge trigger *)
IF in AND NOT edge THEN
	start := TIME();
	IF pt > t#0ms THEN Q := TRUE; END_IF;
END_IF;
edge := in;
IF q THEN
	et := TIME() - start;
	IF et >= PT THEN
		Q := FALSE;
		et := t#0ms;
	END_IF;
END_IF;
END_FUNCTION_BLOCK

(* POU pwm_pw, ST *)
FUNCTION_BLOCK pwm_pw
VAR_INPUT
	F : REAL;
	PW : TIME;
END_VAR
VAR_OUTPUT
	Q : BOOL;
END_VAR
VAR
	clk: CLK_Prg;
	pulse: TP_R;
END_VAR

(*
	version 1.1	25 feb 2007
	programmer 	oscat
	tested BY		oscat

this signal generator generates a square wave signal which is specified by the frequency and the pulse width.
*)
CLK(PT := REAL_TO_TIME(1000/F));
Pulse(in := clk.Q, pt := pw);
Q := pulse.Q;

(* revision history

hm		25. feb 2007	rev 1.1
	recoded in st for better performance and better portability

*)
END_FUNCTION_BLOCK

(* POU Real_To_StrF, ST *)
FUNCTION Real_To_StrF : STRING
VAR_INPUT
	IN : REAL;
	N : INT;
END_VAR
VAR
	dw1 : DWORD;
	dw2 : DWORD;
	s1: STRING;
	s2 : STRING;
END_VAR
dw1 := TRUNC(ABS(in));
dw2 := TRUNC(round(fract(ABS(in))*EXPT(10,N),0));
IF in < 0 THEN
	s1 := CONCAT('-', DWORD_TO_STRING(dw1));
ELSE
	s1 := DWORD_TO_STRING(dw1);
END_IF;
	s1 := CONCAT(s1, '.');
s2 := DWORD_To_STRF(dw2,N);
Real_To_StrF := CONCAT(s1, s2);
END_FUNCTION

(* POU round, ST *)
FUNCTION round : REAL
VAR_INPUT
	in : REAL;
	N : INT;
END_VAR
VAR
END_VAR

(*
version 1.0	1 sep 2006
programmer 	hugo
tested by		tobias

this function rounds a real down to n digits behind the comma.
round(3.1415,1) = 3.1

*)
round := TRUNC(in * EXPT(10,N) + 0.5)/EXPT(10,N);
END_FUNCTION

(* POU Res_NI, ST *)
FUNCTION Res_NI : REAL
VAR_INPUT
	T : REAL;
	R0 : REAL;
END_VAR
VAR CONSTANT
	A : REAL := 0.5485;
	B : REAL := 0.665E-3;
	C : REAL := 2.805E-9;
END_VAR
VAR
END_VAR

(*
version 1.0	4 aug 2006
programmer 	hugo
tested by		tobias

this function returs the resistance for a nickel sensor for a temperature range from -60..+180 °C *)
Res_NI := R0 + A*T + B*EXPT(T,2) + C*EXPT(T,4);



(*

 Auszug aus DIN 43760 für Ni100

°C		R		°C		R		°C	R		°C		R		°C		R

-60 	69,5 	-10 	94,6 	40 	123,0 	90 		154,9 	140 	190,9
-55 	71,9 	-5 		97,3 	45 	126,0 	95 		158,3 	145 	194,8
-50 	74,3 	0 		100,0 	50 	129,1 	100 	161,8 	150 	198,7
-45 	76,7 	5 		102,8 	55 	132,2 	105 	165,3 	155 	202,6
-40 	79,1 	10 		105,6 	60 	135,3 	110 	168,8 	160 	206,6
-35 	81,6 	15 		108,4 	65 	138,5 	115 	172,4 	165 	210,7
-30 	84,2 	20 		111,2 	70 	141,7 	120 	176,0 	170 	214,8
-25 	86,7 	25 		114,1 	75 	145,0 	125 	179,6 	175 	219,0
-20 	89,3 	30 		117,1 	80 	148,3 	130 	183,3 	180 	223,2
-15 	91,9 	35 		120,0 	85 	151,6 	135 	187,1 	  	 

*)
END_FUNCTION

(* POU Res_PT, ST *)
FUNCTION Res_PT : REAL
VAR_INPUT
	T : REAL;
	R0 : REAL;
END_VAR
VAR CONSTANT
	A : REAL := 3.90802E-3 ;
	B : REAL := -5.80195E-7;
	C : REAL := -4.27350E-12;
END_VAR
VAR
END_VAR

(*
version 1.0	4 aug 2006
programmer 	hugo
tested by		tobias


this function returs the resistance for a platinum sensor for a temperature range from -200..+850 °C *)
IF T >= 0 THEN
	Res_PT := R0 * ( 1 + A*T + B*T*T);
ELSE
	Res_PT := R0 * ( 1 + A*T + B*T*T + C*(T-100)*T*T*T);
END_IF;


(*
 Auszug aus DIN 43760 für Pt100

°C		R		°C		R		°C	R			°C		R			°C		R			°C		R

-200 	18,49 	-100 	60,25 	0 	100,00 	100 	138,50 	200 	175,84 	300 	212,02
-195 	20,65 	-95 	62,28 	5 	101,95 	105 	140,39 	205 	177,68 	305 	213,80
-190 	22,80 	-90 	64,30 	10 	103,90 	110 	142,29 	210 	179,51 	310 	215,57
-185 	24,94 	-85 	66,31 	15 	105,85 	115 	144,17 	215 	181,34 	315 	217,35
-180 	27,08 	-80 	68,33 	20 	107,79 	120 	146,06 	220 	183,17 	320 	219,12
-175 	29,20 	-75 	70,33 	25 	109,73 	125 	147,94 	225 	184,99 	325 	220,88
-170 	31,32 	-70 	72,33 	30 	111,67 	130 	149,82 	230 	186,82 	330 	222,65
-165 	33,43 	-65 	74,33 	35 	113,61 	135 	151,70 	235 	188,63 	335 	224,41
-160 	35,33 	-60 	76,33 	40 	115,54 	140 	153,58 	240 	190,45 	340 	226,17
-155 	37,63 	-55 	78,32 	45 	117,47 	145 	155,45 	245 	192,26 	345 	227,92
-150 	39,71 	-50 	80,31 	50 	119,40 	150 	157,31 	250 	194,07 	350 	229,67
-145 	41,79 	-45 	82,29 	55 	121,32 	155 	159,18 	255 	195,88 	355 	231,42
-140 	43,87 	-40 	84,27 	60 	123,24 	160 	161,04 	260 	197,69 	360 	233,17
-135 	45,94 	-35 	86,25 	65 	125,16 	165 	162,90 	265 	199,49 	365 	234,91
-130 	48,00 	-30 	88,22 	70 	127,07 	170 	164,76 	270 	201,29 	370 	236,65
-125 	50,06 	-25 	90,19 	75 	128,98 	175 	166,61 	275 	203,08 	375 	238,39
-120 	52,11 	-20 	92,16 	80 	130,89 	180 	168,46 	280 	204,88 	380 	240,13
-115 	54,15 	-15 	94,12 	85 	132,80 	185 	170,31 	285 	206,67 	385 	241,86
-110 	56,19 	-10 	96,09 	90 	134,70 	190 	172,16 	290 	208,45 	390 	243,59
-105 	58,22 	-5 		98,04 	95 	136,60 	195 	174,00 	295 	210,24 	395 	245,31

*)
END_FUNCTION

(* POU Res_SI, ST *)
FUNCTION Res_SI : REAL
VAR_INPUT
	T : REAL;
	RS : REAL;
	TS : REAL;
END_VAR
VAR CONSTANT
	A : REAL := 7.64E-3;
	B : REAL := 1.66E-5;
END_VAR
VAR
END_VAR

(*
version 1.0	4 aug 2006
programmer 	hugo
tested by		tobias

this function returs the resistance for a silicon sensor for a temperature range from -50..+150 °C
for example KTY10 normaly Rs at 25 °C
*)
Res_SI := RS * ( 1 + A * (T - TS) + B * EXPT(T - TS, 2));
END_FUNCTION

(* POU rmp_B, ST *)
FUNCTION_BLOCK rmp_B
VAR_INPUT
	SET : BOOL := FALSE;
	PT : TIME;
	EN : BOOL := TRUE;
	UP : BOOL := TRUE;
	RST : BOOL := FALSE;
END_VAR
VAR_OUTPUT
	Out : BYTE := 0;
	busy: BOOL;
END_VAR
VAR
	last_step : TIME := T#0ms;
	now : TIME;
END_VAR

(*
	version 1.2	17 jan 2007
	programmer 	oscat
	tested BY		oscat

this ramp generator generates a byte wide ramp with 255 steps
the generator has an asynchronous set and reset
the ramp is controlled by PT which is the total ramp time for a full sweep from 0..255
an UD input controlls the direction Up or Down and the E input enables the ramp generation
a busy output indicates that the ramp is running, busy false means output is stable.

*)
IF en  THEN
	(* generate ramp *)
	now := TIME();
	IF now >= last_step + pt / 255 THEN
		last_step := now;
		IF UP AND out < 255 THEN out := out + 1; END_IF;
		IF NOT UP AND out > 0 THEN out := out -1; END_IF;
	END_IF;
END_IF;

(* check for asynchronous set or reset *)
IF set  THEN out := 255; END_IF;
IF rst THEN out := 0; END_IF;

(* checks for outputs stable and reset or set busy flag *)
IF out = 0 OR out = 255 THEN busy := FALSE; ELSE busy := TRUE; END_IF;

(* revision history

hm 5.10.2006	rev 1.1
	added busy output
hm 17.1.2007	rev 1.2
	renamed input ud to up for better usability
	deleted unused variable step

*)
END_FUNCTION_BLOCK

(* POU rmp_soft, ST *)
FUNCTION_BLOCK rmp_soft
VAR_INPUT
	IN : BOOL;
	val : BYTE;
END_VAR
VAR_INPUT CONSTANT
	pt_on: TIME := T#100ms;
	PT_off : TIME := T#100ms;
END_VAR
VAR CONSTANT
	steps : INT := 255;
END_VAR
VAR_OUTPUT
	Out : BYTE := 0;
END_VAR
VAR
	last_step : TIME := T#0ms;
	now : TIME;
	x :REAL := 0;
END_VAR

(*
	version 1.0	22 jan 2007
	programmer 	oscat
	tested BY		oscat

this soft on/off ramp generator generates a soft on and soft off ramp while the max on value is set by the input
the time for a full ramp can be set by config variables for up and down ramp.
*)
IF in  AND out < val THEN
	(* generate on ramp *)
	now := TIME();
	x := out + TIME_TO_REAL(now -last_step)*steps/TIME_TO_REAL(pt_on);
	IF x > val THEN
		out := val;
		x := val;
	ELSE out := REAL_TO_BYTE(x); END_IF;
	last_step := now;
ELSIF NOT in AND out > 0 THEN
	(* generate off ramp *)
	now := TIME();
	x := out - TIME_TO_REAL(now -last_step)*steps/TIME_TO_REAL(pt_off);
	IF x  < 0 THEN
		out := 0;
		x := 0;
	ELSE out := REAL_TO_BYTE(x); END_IF;
	last_step := now;
ELSIF in AND out > val THEN
	(* generate ramp down to input value *)
	now := TIME();
	x := out - TIME_TO_REAL(now -last_step)*steps/TIME_TO_REAL(pt_off);
	IF x  < val THEN
		out := val;
		x := val;
	ELSE out := REAL_TO_BYTE(x); END_IF;
	last_step := now;
END_IF;
IF out = val OR out = 0 THEN last_step := TIME(); END_IF;


(* revision history

hm 22.1.2007		rev 1.1
	deleted unused variables X1 and I, X2 and X3

*)
END_FUNCTION_BLOCK

(* POU rmp_W, ST *)
FUNCTION_BLOCK rmp_W
VAR_INPUT
	SET : BOOL := FALSE;
	PT : TIME;
	EN : BOOL := TRUE;
	UD : BOOL := TRUE;
	RST : BOOL := FALSE;
END_VAR
VAR_OUTPUT
	Out : WORD := 0;
	busy : BOOL;
END_VAR
VAR
	last_step : TIME := T#0ms;
	now : TIME;
END_VAR

(*
	version 1.2	22 Jan 2007
	programmer 	oscat
	tested BY		oscat

this ramp generator generates a Word wide ramp with 65535 steps
the generator has an asynchronous set and reset
the ramp is controlled by PT which is the total ramp time for a full sweep from 0..65535
an UD input controlls the direction Up or Down and the E input enables the ramp generation
a busy output indicates that the ramp is running, busy false means output is stable.
*)
IF en  THEN
	(* generate ramp *)
	now := TIME();
	IF now >= last_step + pt / 65535 THEN
		last_step := now;
		IF UD AND out < 65535 THEN out := out + 1; END_IF;
		IF NOT ud AND out > 0 THEN out := out -1; END_IF;
	END_IF;
END_IF;

(* check for asynchronous set or reset *)
IF set  THEN out := 65535; END_IF;
IF rst THEN out := 0; END_IF;

(* set or reset the busy flag *)
IF out = 0 OR out = 65535 THEN busy := FALSE; ELSE busy := TRUE; END_IF;

(* revision history:

hm 4.10.2006		rev 1.1
	added the busy output which signals that the ramp is running.

hm 22.1.2007		rev 1.2
	deleted unused variable step

*)
END_FUNCTION_BLOCK

(* POU scale_B2, ST *)
FUNCTION scale_B2 : REAL
VAR_INPUT
	in1: BYTE;
	in2: BYTE;
	K : REAL := 1;
	O : REAL := 0;
END_VAR
VAR_INPUT CONSTANT
	in1_min: REAL := 0;
	in1_max: REAL := 1000;
	in2_min: REAL := 0;
	in2_max: REAL := 1000;
END_VAR

(*
version 1.1	19 jan 2007
programmer 	hugo
tested by		tobias

	this functiob block can scale up to two inputs.
	the inputs have their min value at 0 and their max value at 255 while the min and max value can be either positive or negative.
	the inputs ramp between min and max values for the respective inputs to be between (0..255).
	the summed output is then scaled by an scale input K and a offset O can be added to the output.
	the min and max input configurations can be edited in the cfc editor by double clicking the symbol body.

*)
scale_B2 := 	((in1_max - in1_min)* in1 / 255 + in1_min +
				(in2_max - in2_min)* in2 / 255 + in2_min)
				* K + O;

(* revision History
hm 19.1.2007	rev 1.1
	changed outputs to real to avoid overflow of integer
	added offset for better cascading of scale functions
	changed from FB to function
*)
END_FUNCTION

(* POU scale_B4, ST *)
FUNCTION scale_B4 : REAL
VAR_INPUT
	in1: BYTE;
	in2: BYTE;
	in3: BYTE;
	in4: BYTE;
	K : REAL := 1;
	O : REAL := 0;
END_VAR
VAR_INPUT CONSTANT
	in1_min: REAL := 0;
	in1_max: REAL := 1000;
	in2_min: REAL := 0;
	in2_max: REAL := 1000;
	in3_min: REAL := 0;
	in3_max: REAL := 1000;
	in4_min: REAL := 0;
	in4_max: REAL := 1000;
END_VAR

(*
version 1.1	19 jan 2007
programmer 	hugo
tested by		tobias

	this functiob block can scale up to 4 inputs.
	the inputs have their min value at 0 and their max value at 255 while the min and max value can be either positive or negative.
	the inputs ramp between min and max values for the respective inputs to be between (0..255).
	the summed output is then scaled by an scale input K and a offset O can be added to the output.
	the min and max input configurations can be edited in the cfc editor by double clicking the symbol body.

*)
scale_B4 := 	((in1_max - in1_min)* in1 / 255 + in1_min +
				(in2_max - in2_min)* in2 / 255 + in2_min +
				(in3_max - in3_min)* in3 / 255 + in3_min +
				(in4_max - in4_min)* in4 / 255 + in4_min)
				* K + O;

(* revision History
hm 19.1.2007	rev 1.1
	changed outputs to real to avoid overflow of integer
	added offset for better cascading of scale functions
	changed from fb to function
*)
END_FUNCTION

(* POU scale_B8, ST *)
FUNCTION scale_B8 : REAL
VAR_INPUT
	in1: BYTE;
	in2: BYTE;
	in3: BYTE;
	in4: BYTE;
	in5: BYTE;
	in6: BYTE;
	in7: BYTE;
	in8: BYTE;
	K : REAL := 1;
	O : REAL := 0;
END_VAR
VAR_INPUT CONSTANT
	in1_min: REAL := 0;
	in1_max: REAL := 1000;
	in2_min: REAL := 0;
	in2_max: REAL := 1000;
	in3_min: REAL := 0;
	in3_max: REAL := 1000;
	in4_min: REAL := 0;
	in4_max: REAL := 1000;
	in5_min: REAL := 0;
	in5_max: REAL := 1000;
	in6_min: REAL := 0;
	in6_max: REAL := 1000;
	in7_min: REAL := 0;
	in7_max: REAL := 1000;
	in8_min: REAL := 0;
	in8_max: REAL := 1000;
END_VAR

(*
version 1.1	19 jan 2007
programmer 	hugo
tested by		tobias

	this functiob block can scale up to 8 inputs.
	the inputs have their min value at 0 and their max value at 255 while the min and max value can be either positive or negative.
	the inputs ramp between min and max values for the respective inputs to be between (0..255).
	the summed output is then scaled by an scale input K and a offset O can be added to the output.
	the min and max input configurations can be edited in the cfc editor by double clicking the symbol body.

*)
scale_B8 := 	((in1_max - in1_min)* in1 / 255 + in1_min +
				(in2_max - in2_min)* in2 / 255 + in2_min +
				(in3_max - in3_min)* in3 / 255 + in3_min +
				(in4_max - in4_min)* in4 / 255 + in4_min +
				(in5_max - in5_min)* in5 / 255 + in5_min +
				(in6_max - in6_min)* in6 / 255 + in6_min +
				(in7_max - in7_min)* in7 / 255 + in7_min +
				(in8_max - in8_min)* in8 / 255 + in8_min)
				* K + O;

(* revision History
hm 19.1.2007	rev 1.1
	changed outputs to real to avoid overflow of integer
	added offset for better cascading of scale functions
*)
END_FUNCTION

(* POU scale_X2, ST *)
FUNCTION scale_X2 : REAL
VAR_INPUT
	in1: BOOL;
	in2: BOOL;
	K : REAL := 1;
	O : REAL := 0;
END_VAR
VAR_INPUT CONSTANT
	in1_min: REAL := 0;
	in1_max: REAL := 1000;
	in2_min: REAL := 0;
	in2_max: REAL := 1000;
END_VAR

(*
version 1.0	19 jan 2007
programmer 	hugo
tested by		tobias

	this functiob block can scale up to two inputs.
	the input can select between two ues with true or false.
	the summed output is then scaled by an scale input K and a offset O can be added to the output.
	the min and max input configurations can be edited in the cfc editor by double clicking the symbol body.

*)
IF NOT in1 THEN scale_x2 := in1_min; ELSE scale_x2 := in1_max; END_IF;
IF NOT in2 THEN scale_x2 := scale_x2 + in2_min; ELSE scale_x2 := scale_x2 + in2_max; END_IF;
scale_X2 := scale_X2 * k + O;

(* revision history

*)
END_FUNCTION

(* POU scale_X4, ST *)
FUNCTION scale_X4 : REAL
VAR_INPUT
	in1: BOOL;
	in2: BOOL;
	in3: BOOL;
	in4: BOOL;
	K : REAL := 1;
	O : REAL := 0;
END_VAR
VAR_INPUT CONSTANT
	in1_min: REAL := 0;
	in1_max: REAL := 1000;
	in2_min: REAL := 0;
	in2_max: REAL := 1000;
	in3_min: REAL := 0;
	in3_max: REAL := 1000;
	in4_min: REAL := 0;
	in4_max: REAL := 1000;
END_VAR

(*
version 1.0	19 jan 2007
programmer 	hugo
tested by		tobias

	this function can scale up to 4 inputs.
	the input can select between two ues with true or false.
	the summed output is then scaled by an scale input K and a offset O can be added to the output.
	the min and max input configurations can be edited in the cfc editor by double clicking the symbol body.

*)
IF NOT in1 THEN scale_X4 := in1_min; ELSE scale_X4 := in1_max; END_IF;
IF NOT in2 THEN scale_x4 := scale_x4 + in2_min; ELSE scale_x4 := scale_x4 + in2_max; END_IF;
IF NOT in3 THEN scale_x4 := scale_x4 + in3_min; ELSE scale_x4 := scale_x4 + in3_max; END_IF;
IF NOT in4 THEN scale_x4 := scale_x4 + in4_min; ELSE scale_x4 := scale_x4 + in4_max; END_IF;
scale_X4 := scale_X4 * k + O;

(* revision history

*)
END_FUNCTION

(* POU scale_X8, ST *)
FUNCTION scale_X8 : REAL
VAR_INPUT
	in1: BOOL;
	in2: BOOL;
	in3: BOOL;
	in4: BOOL;
	in5: BOOL;
	in6: BOOL;
	in7: BOOL;
	in8: BOOL;
	K : REAL := 1;
	O : REAL := 0;
END_VAR
VAR_INPUT CONSTANT
	in1_min: REAL := 0;
	in1_max: REAL := 1000;
	in2_min: REAL := 0;
	in2_max: REAL := 1000;
	in3_min: REAL := 0;
	in3_max: REAL := 1000;
	in4_min: REAL := 0;
	in4_max: REAL := 1000;
	in5_min: REAL := 0;
	in5_max: REAL := 1000;
	in6_min: REAL := 0;
	in6_max: REAL := 1000;
	in7_min: REAL := 0;
	in7_max: REAL := 1000;
	in8_min: REAL := 0;
	in8_max: REAL := 1000;
END_VAR

(*
version 1.0	19 jan 2007
programmer 	hugo
tested by		tobias

	this function can scale up to 4 inputs.
	the input can select between two ues with true or false.
	the summed output is then scaled by an scale input K and a offset O can be added to the output.
	the min and max input configurations can be edited in the cfc editor by double clicking the symbol body.

*)
IF NOT in1 THEN scale_x8 := in1_min; ELSE scale_x8 := in1_max; END_IF;
IF NOT in2 THEN scale_x8 := scale_x8 + in2_min; ELSE scale_x8 := scale_x8 + in2_max; END_IF;
IF NOT in3 THEN scale_x8 := scale_x8 + in3_min; ELSE scale_x8 := scale_x8 + in3_max; END_IF;
IF NOT in4 THEN scale_x8 := scale_x8 + in4_min; ELSE scale_x8 := scale_x8 + in4_max; END_IF;
IF NOT in5 THEN scale_x8 := scale_x8 + in5_min; ELSE scale_x8 := scale_x8 + in5_max; END_IF;
IF NOT in6 THEN scale_x8 := scale_x8 + in6_min; ELSE scale_x8 := scale_x8 + in6_max; END_IF;
IF NOT in7 THEN scale_x8 := scale_x8 + in7_min; ELSE scale_x8 := scale_x8 + in7_max; END_IF;
IF NOT in8 THEN scale_x8 := scale_x8 + in8_min; ELSE scale_x8 := scale_x8 + in8_max; END_IF;
scale_X8 := scale_X8 * k + O;

(* revision history

*)
END_FUNCTION

(* POU second_to_time, ST *)
FUNCTION second_to_time : TIME
VAR_INPUT
	input : REAL;
END_VAR
VAR
END_VAR

(*
version 1.0	4 aug 2006
programmer 	hugo
tested by		tobias

converts an amount of seconds in real to time
execution TIME on wago 750-841 =  17us 

*)
second_to_time := DWORD_TO_TIME(REAL_TO_DWORD(input * 1000));
END_FUNCTION

(* POU Sensor_Int, ST *)
FUNCTION Sensor_Int : REAL
VAR_INPUT
	Voltage : REAL;
	Current : REAL;
	RP : REAL;
	RS : REAL;
END_VAR
VAR
	Rx: REAL;
END_VAR

(*
version 1.1	20 jan 2007
programmer 	hugo
tested by		tobias

this function calculates the real resistance of a sensor RX given a parasitic resistor in parallel to the sensor and an additional serial resistor.
for example a parasitic parallel resistor for a PT100 can be ignored but a series resistor is the cable to the sensor.
for a humidity sensor, the parallel resistor is more dramatic and needs to be considered.
the function allows to consider a parallel and serial resistor at the same time.
with this function and known parasitic serial and parallel resistors the true resistance of the sensor can be calculated.

*)
Rx := RP * ( voltage / current - RS) / ( RP + RS - Voltage / Current);

(* revisaion history

hm 20.1.2007	rev 1.1
	deleted input R0 which was not needed.

*)
END_FUNCTION

(* POU sequence_4, ST *)
FUNCTION_BLOCK sequence_4
VAR_INPUT
	in0 : BOOL := TRUE;
	in1 : BOOL := TRUE;
	in2 : BOOL := TRUE;
	in3 : BOOL := TRUE;
	start : BOOL;
	rst : BOOL;
	wait0 : TIME := t#0s;
	delay0 : TIME := t#0s;
	wait1 : TIME := t#0s;
	delay1 : TIME := t#0s;
	wait2 : TIME := t#0s;
	delay2 : TIME := t#0s;
	wait3 : TIME := t#0s;
	delay3 : TIME := t#0s;
END_VAR
VAR_INPUT CONSTANT
	stop_on_error : BOOL := FALSE;
END_VAR
VAR_OUTPUT
	Q0 : BOOL;
	Q1 : BOOL;
	Q2 : BOOL;
	Q3 : BOOL;
	any : BOOL;
	run: BOOL;
	step : INT := -1;
	status : BYTE := 0;
END_VAR
VAR
	last : TIME;
	edge : BOOL;
	tx: TIME;
	init: BOOL;
END_VAR

(*
version 1.3	17 jan 2007
programmer 	oscat
tested by		hans

sequence_4 enables run when a low to high transition is present on start.
a low to high transition on start will restart the sequencer at any time while a rst will hold the sequencer in reset while true.
after run is enabled with a rising edge on start the sequencer waits for wait0 on in0 to enable q0 which stays on for delay0.
the next cycle starts with wait1, continues with delay 1 and so on...
if an edge is not detected during the wait period, the sequencer will then display the error number on the status output.
the status numbers 1..4 are errors in step 0..3.
after the last step that sets q3, the sequencer leaves q3 on for delay3 and then resets to the initial state.
a step output will indicate the current step of the sequencer and will also be present with a fault condition.
after the first output is turened on the sequencer switches from q0 to q1 and so on, at any time there is only one output enabled.
if an input signal is not detected during a wait period, the sequencer will display the error number ( 1 for in0, 2 for in1 .... ).
when an error is present and the config variable stop_on_error is set then the sequencer will stop. otherwise it will continue.
The status output will also display 110 for waiting and 111 for sequence running.
*)
(* read sps timer *)
tx := TIME();

(* initialize on startup *)
IF NOT init THEN
	last := tx;
	init := TRUE;
	status := 110;
END_IF;

(* asynchronous reset *)
IF rst THEN
	step := -1;
	Q0 := 0;
	Q1 := 0;
	Q2 := 0;
	Q3 := 0;
	status := 110;
	run := 0;

(* edge on start input restarts the sequencer *)
ELSIF start AND NOT edge THEN
	step := 0;
	last := tx;
	status := 111;
	Q0 := 0;
	Q1 := 0;
	Q2 := 0;
	Q3 := 0;
	run := 1;
END_IF;
edge := start;

(* check if stop on status is necessary *)
IF status > 0 AND status < 100 AND stop_on_error THEN RETURN; END_IF;

(* sequence is running *)
IF run AND step = 0 THEN
	IF NOT q0 AND in0 AND tx - last <= wait0 THEN
		Q0 := TRUE;
		last := tx;
	ELSIF NOT q0 AND tx - last > wait0 THEN
		status := 1;
		run := FALSE;
	ELSIF q0 AND tx - last >= delay0 THEN
		step := 1;
		last := tx;
	END_IF;
END_IF;
IF run AND step = 1 THEN
	IF NOT q1 AND in1 AND tx - last <= wait1 THEN
		Q0 := FALSE;
		Q1 := TRUE;
		last := tx;
	ELSIF NOT q1 AND Tx - last > wait1 THEN
		status := 2;
		q0 := FALSE;
		run := FALSE;
	ELSIF q1 AND tx - last >= delay1 THEN
		step := 2;
		last := tx;
	END_IF;
END_IF;
IF run AND step = 2 THEN
	IF NOT q2 AND in2 AND tx - last <= wait2 THEN
		Q1 := FALSE;
		Q2 := TRUE;
		last := tx;
	ELSIF NOT q2 AND Tx - last > wait2 THEN
		status := 3;
		q1 := FALSE;
		run := FALSE;
	ELSIF q2 AND tx - last >= delay2 THEN
		step := 3;
		last := tx;
	END_IF;
END_IF;
IF run AND step = 3 THEN
	IF NOT q3 AND in3 AND tx - last <= wait3 THEN
		Q2 := FALSE;
		Q3 := TRUE;
		last := tx;
	ELSIF NOT q3 AND Tx - last > wait3 THEN
		status := 4;
		q2 := FALSE;
		run := FALSE;
	ELSIF q3 AND tx - last >= delay3 THEN
		step := -1;
		q3 := FALSE;
		run := FALSE;
		status := 110;
	END_IF;
END_IF;
any := q0 OR q1 OR q2 OR q3;

(*
hm 1.10.06		rev 1.1
	corrected delay logic to be after event and not before
	added any output

hm 1.12.06		rev 1.2
	corrected failure in sequence logic.
	added init at startup to prevent from initial statuss after start.

hm 17.1.2007		rev 1.3
	changed output fault to status for better compatibility with other modules (ESR).
	added stop on error functionality and setup variable
	default for inputs in0..3 is true.
	renamed variable state to step
*)
END_FUNCTION_BLOCK

(* POU set_Tod, ST *)
FUNCTION set_Tod : TOD
VAR_INPUT
	hour : INT;
	minute : INT;
	second : REAL;
END_VAR
VAR
END_VAR

(*
version 1.0	4 aug 2006
programmer 	hugo
tested by		tobias

creates tod from hour minute and second 
execution time on wago 750-841 = 14 us  
*)
set_Tod := DWORD_TO_TOD(TRUNC(second * 1000) + minute * 60000 + hour * 3600000);
END_FUNCTION

